LIN {X 0,Y 282.516,Z 595.13,A -85,B 0,C 180,E1 -17100,E2 -17100} C_VEL
LIN {X 0,Y 282.582,Z 591.794,A -85,B 0,C 180,E1 -17102.851,E2 -17102.851} C_VEL
LIN {X 0,Y 282.699,Z 588.163,A -85,B 0,C 180,E1 -17104.992,E2 -17104.992} C_VEL
LIN {X 0,Y 282.973,Z 582.873,A -85,B 0,C 180,E1 -17107.372,E2 -17107.372} C_VEL
LIN {X 0,Y 283.496,Z 576.551,A -85,B 0,C 180,E1 -17109.633,E2 -17109.633} C_VEL
LIN {X 0,Y 284.235,Z 569.125,A -85,B 0,C 180,E1 -17111.771,E2 -17111.771} C_VEL
LIN {X 0,Y 285.228,Z 560.039,A -85,B 0,C 180,E1 -17113.901,E2 -17113.901} C_VEL
LIN {X 0,Y 286.392,Z 549.973,A -85,B 0,C 180,E1 -17115.843,E2 -17115.843} C_VEL
LIN {X 0,Y 287.513,Z 540.083,A -85,B 0,C 180,E1 -17117.419,E2 -17117.419} C_VEL
LIN {X 0,Y 289.014,Z 526.644,A -85,B 0,C 180,E1 -17119.165,E2 -17119.165} C_VEL
LIN {X 0,Y 289.369,Z 520.172,A -85,B 0,C 180,E1 -17119.878,E2 -17119.878} C_VEL
LIN {X 0,Y 287.114,Z 506.341,A -85,B 0,C 180,E1 -17121.272,E2 -17121.272} C_VEL
LIN {X 0,Y 284.752,Z 492.339,A -85,B 0,C 180,E1 -17122.392,E2 -17122.392} C_VEL
LIN {X 0,Y 283.421,Z 484.414,A -85,B 0,C 180,E1 -17122.941,E2 -17122.941} C_VEL
LIN {X 0,Y 283.819,Z 479.195,A -85,B 0,C 180,E1 -17126.942,E2 -17126.942} C_VEL
LIN {X 0,Y 284.155,Z 475.25,A -85,B 0,C 180,E1 -17130.04,E2 -17130.04} C_VEL
LIN {X 0,Y 284.561,Z 470.604,A -85,B 0,C 180,E1 -17133.759,E2 -17133.759} C_VEL
LIN {X 0,Y 284.674,Z 467.49,A -85,B 0,C 180,E1 -17136.336,E2 -17136.336} C_VEL
LIN {X 0,Y 284.462,Z 463.675,A -85,B 0,C 180,E1 -17139.623,E2 -17139.623} C_VEL
LIN {X 0,Y 284.349,Z 463.813,A -85,B 0,C 180,E1 -17141.152,E2 -17141.152} C_VEL
LIN {X 0,Y 285.36,Z 468.719,A -85,B 0,C 180,E1 -17144.418,E2 -17144.418} C_VEL
LIN {X 0,Y 286.241,Z 473.395,A -85,B 0,C 180,E1 -17147.441,E2 -17147.441} C_VEL
LIN {X 0,Y 286.899,Z 478.224,A -85,B 0,C 180,E1 -17150.437,E2 -17150.437} C_VEL
LIN {X 0,Y 286.537,Z 484.384,A -85,B 0,C 180,E1 -17153.937,E2 -17153.937} C_VEL
LIN {X 0,Y 285.97,Z 492.07,A -85,B 0,C 180,E1 -17158.103,E2 -17158.103} C_VEL
LIN {X 0,Y 285.889,Z 493.182,A -85,B 0,C 180,E1 -17158.662,E2 -17158.662} C_VEL
LIN {X 0,Y 290.88,Z 508.242,A -85,B 0,C 180,E1 -17159.827,E2 -17159.827} C_VEL
LIN {X 0,Y 294.37,Z 521.693,A -85,B 0,C 180,E1 -17161.017,E2 -17161.017} C_VEL
LIN {X 0,Y 296.863,Z 535.081,A -85,B 0,C 180,E1 -17162.363,E2 -17162.363} C_VEL
LIN {X 0,Y 297.951,Z 545.247,A -85,B 0,C 180,E1 -17163.511,E2 -17163.511} C_VEL
LIN {X 0,Y 296.029,Z 557.79,A -85,B 0,C 180,E1 -17164.888,E2 -17164.888} C_VEL
LIN {X 0,Y 293.603,Z 570.03,A -85,B 0,C 180,E1 -17166.548,E2 -17166.548} C_VEL
LIN {X 0,Y 291.679,Z 579.114,A -85,B 0,C 180,E1 -17168.068,E2 -17168.068} C_VEL
LIN {X 0,Y 289.463,Z 589.297,A -85,B 0,C 180,E1 -17170.127,E2 -17170.127} C_VEL
LIN {X 0,Y 287.506,Z 597.701,A -85,B 0,C 180,E1 -17172.207,E2 -17172.207} C_VEL
LIN {X 0,Y 285.969,Z 605.714,A -85,B 0,C 180,E1 -17174.679,E2 -17174.679} C_VEL
LIN {X 0,Y 284.396,Z 612.165,A -85,B 0,C 180,E1 -17177.148,E2 -17177.148} C_VEL
LIN {X 0,Y 283.335,Z 617.873,A -85,B 0,C 180,E1 -17179.999,E2 -17179.999} C_VEL
LIN {X 0,Y 282.7,Z 622.021,A -85,B 0,C 180,E1 -17182.858,E2 -17182.858} C_VEL
LIN {X 0,Y 282.371,Z 624.74,A -85,B 0,C 180,E1 -17185.716,E2 -17185.716} C_VEL
LIN {X 0,Y 282.307,Z 626.104,A -85,B 0,C 180,E1 -17188.572,E2 -17188.572} C_VEL
LIN {X 0,Y 282.307,Z 626.137,A -85,B 0,C 180,E1 -17191.425,E2 -17191.425} C_VEL
LIN {X 0,Y 282.369,Z 624.833,A -85,B 0,C 180,E1 -17194.28,E2 -17194.28} C_VEL
LIN {X 0,Y 282.697,Z 622.169,A -85,B 0,C 180,E1 -17197.139,E2 -17197.139} C_VEL
LIN {X 0,Y 283.317,Z 618.072,A -85,B 0,C 180,E1 -17199.998,E2 -17199.998} C_VEL
LIN {X 0,Y 284.328,Z 612.422,A -85,B 0,C 180,E1 -17202.852,E2 -17202.852} C_VEL
LIN {X 0,Y 285.9,Z 606.036,A -85,B 0,C 180,E1 -17205.321,E2 -17205.321} C_VEL
LIN {X 0,Y 287.441,Z 598.344,A -85,B 0,C 180,E1 -17207.72,E2 -17207.72} C_VEL
LIN {X 0,Y 289.392,Z 589.781,A -85,B 0,C 180,E1 -17209.875,E2 -17209.875} C_VEL
LIN {X 0,Y 291.625,Z 579.728,A -85,B 0,C 180,E1 -17211.932,E2 -17211.932} C_VEL
LIN {X 0,Y 293.983,Z 568.473,A -85,B 0,C 180,E1 -17213.79,E2 -17213.79} C_VEL
LIN {X 0,Y 296.157,Z 557.289,A -85,B 0,C 180,E1 -17215.285,E2 -17215.285} C_VEL
LIN {X 0,Y 298.037,Z 545.082,A -85,B 0,C 180,E1 -17216.616,E2 -17216.616} C_VEL
LIN {X 0,Y 296.515,Z 532.609,A -85,B 0,C 180,E1 -17218.007,E2 -17218.007} C_VEL
LIN {X 0,Y 293.649,Z 518.477,A -85,B 0,C 180,E1 -17219.397,E2 -17219.397} C_VEL
LIN {X 0,Y 290.039,Z 505.316,A -85,B 0,C 180,E1 -17220.528,E2 -17220.528} C_VEL
LIN {X 0,Y 285.892,Z 493.075,A -85,B 0,C 180,E1 -17221.49,E2 -17221.49} C_VEL
LIN {X 0,Y 286.527,Z 484.62,A -85,B 0,C 180,E1 -17226.061,E2 -17226.061} C_VEL
LIN {X 0,Y 286.962,Z 478.474,A -85,B 0,C 180,E1 -17229.548,E2 -17229.548} C_VEL
LIN {X 0,Y 286.339,Z 473.573,A -85,B 0,C 180,E1 -17232.58,E2 -17232.58} C_VEL
LIN {X 0,Y 285.25,Z 467.689,A -85,B 0,C 180,E1 -17236.38,E2 -17236.38} C_VEL
LIN {X 0,Y 284.343,Z 463.696,A -85,B 0,C 180,E1 -17239.081,E2 -17239.081} C_VEL
LIN {X 0,Y 284.347,Z 463.691,A -85,B 0,C 180,E1 -17243.616,E2 -17243.616} C_VEL
LIN {X 0,Y 284.301,Z 463.7,A -85,B 0,C 180,E1 -17247.188,E2 -17247.188} C_VEL
LIN {X 0,Y 284.354,Z 463.689,A -85,B 0,C 180,E1 -17250.375,E2 -17250.375} C_VEL
LIN {X 0,Y 284.371,Z 463.676,A -85,B 0,C 180,E1 -17253.586,E2 -17253.586} C_VEL
LIN {X 0,Y 284.366,Z 463.681,A -85,B 0,C 180,E1 -17256.707,E2 -17256.707} C_VEL
LIN {X 0,Y 284.421,Z 463.678,A -85,B 0,C 180,E1 -17259.873,E2 -17259.873} C_VEL
LIN {X 0,Y 284.482,Z 463.671,A -85,B 0,C 180,E1 -17264.458,E2 -17264.458} C_VEL
LIN {X 0,Y 284.48,Z 463.669,A -85,B 0,C 180,E1 -17268.601,E2 -17268.601} C_VEL
LIN {X 0,Y 284.647,Z 463.647,A -85,B 0,C 180,E1 -17271.547,E2 -17271.547} C_VEL
LIN {X 0,Y 283.962,Z 463.739,A -85,B 0,C 180,E1 -17272.726,E2 -17272.726} C_VEL
LIN {X 0,Y 281.114,Z 464.091,A -85,B 0,C 180,E1 -17274.649,E2 -17274.649} C_VEL
LIN {X 0,Y 278.747,Z 464.389,A -85,B 0,C 180,E1 -17276.21,E2 -17276.21} C_VEL
LIN {X 0,Y 277.785,Z 464.506,A -85,B 0,C 180,E1 -17277.419,E2 -17277.419} C_VEL
LIN {X 0,Y 277.735,Z 464.509,A -85,B 0,C 180,E1 -17277.828,E2 -17277.828} C_VEL
LIN {X 0,Y 277.884,Z 464.496,A -85,B 0,C 180,E1 -17280,E2 -17280} C_VEL
LIN {X 0,Y 277.69,Z 464.494,A -85,B 0,C 180,E1 -17282.901,E2 -17282.901} C_VEL
LIN {X 0,Y 277.643,Z 464.526,A -85,B 0,C 180,E1 -17287.271,E2 -17287.271} C_VEL
LIN {X 0,Y 277.497,Z 464.516,A -85,B 0,C 180,E1 -17290.212,E2 -17290.212} C_VEL
LIN {X 0,Y 277.425,Z 464.553,A -85,B 0,C 180,E1 -17294.675,E2 -17294.675} C_VEL
LIN {X 0,Y 277.334,Z 464.554,A -85,B 0,C 180,E1 -17299.234,E2 -17299.234} C_VEL
LIN {X 0,Y 277.31,Z 464.567,A -85,B 0,C 180,E1 -17304.171,E2 -17304.171} C_VEL
LIN {X 0,Y 277.316,Z 464.565,A -85,B 0,C 180,E1 -17307.506,E2 -17307.506} C_VEL
LIN {X 0,Y 277.263,Z 464.572,A -85,B 0,C 180,E1 -17310.482,E2 -17310.482} C_VEL
LIN {X 0,Y 277.246,Z 464.573,A -85,B 0,C 180,E1 -17313.896,E2 -17313.896} C_VEL
LIN {X 0,Y 277.283,Z 464.572,A -85,B 0,C 180,E1 -17317.467,E2 -17317.467} C_VEL
LIN {X 0,Y 277.257,Z 464.571,A -85,B 0,C 180,E1 -17321.228,E2 -17321.228} C_VEL
LIN {X 0,Y 277.308,Z 464.597,A -85,B 0,C 180,E1 -17323.679,E2 -17323.679} C_VEL
LIN {X 0,Y 278.483,Z 471.133,A -85,B 0,C 180,E1 -17328.07,E2 -17328.07} C_VEL
LIN {X 0,Y 279.695,Z 477.445,A -85,B 0,C 180,E1 -17332.088,E2 -17332.088} C_VEL
LIN {X 0,Y 280.717,Z 483.391,A -85,B 0,C 180,E1 -17335.709,E2 -17335.709} C_VEL
LIN {X 0,Y 280.667,Z 484.37,A -85,B 0,C 180,E1 -17336.18,E2 -17336.18} C_VEL
LIN {X 0,Y 280.949,Z 492.018,A -85,B 0,C 180,E1 -17338.069,E2 -17338.069} C_VEL
LIN {X 0,Y 285.484,Z 507.635,A -85,B 0,C 180,E1 -17339.137,E2 -17339.137} C_VEL
LIN {X 0,Y 288.26,Z 521.704,A -85,B 0,C 180,E1 -17340.206,E2 -17340.206} C_VEL
LIN {X 0,Y 290.029,Z 534.468,A -85,B 0,C 180,E1 -17341.351,E2 -17341.351} C_VEL
LIN {X 0,Y 291.046,Z 547.26,A -85,B 0,C 180,E1 -17342.693,E2 -17342.693} C_VEL
LIN {X 0,Y 290.475,Z 552.892,A -85,B 0,C 180,E1 -17343.276,E2 -17343.276} C_VEL
LIN {X 0,Y 288.548,Z 564.116,A -85,B 0,C 180,E1 -17344.577,E2 -17344.577} C_VEL
LIN {X 0,Y 286.145,Z 576.029,A -85,B 0,C 180,E1 -17346.287,E2 -17346.287} C_VEL
LIN {X 0,Y 283.762,Z 586.747,A -85,B 0,C 180,E1 -17348.193,E2 -17348.193} C_VEL
LIN {X 0,Y 281.559,Z 596.39,A -85,B 0,C 180,E1 -17350.31,E2 -17350.31} C_VEL
LIN {X 0,Y 279.68,Z 604.372,A -85,B 0,C 180,E1 -17352.452,E2 -17352.452} C_VEL
LIN {X 0,Y 278.313,Z 611.004,A -85,B 0,C 180,E1 -17354.626,E2 -17354.626} C_VEL
LIN {X 0,Y 277.137,Z 616.5,A -85,B 0,C 180,E1 -17356.809,E2 -17356.809} C_VEL
LIN {X 0,Y 276.088,Z 622.251,A -85,B 0,C 180,E1 -17359.738,E2 -17359.738} C_VEL
LIN {X 0,Y 275.484,Z 626.427,A -85,B 0,C 180,E1 -17362.673,E2 -17362.673} C_VEL
LIN {X 0,Y 275.242,Z 629.15,A -85,B 0,C 180,E1 -17365.609,E2 -17365.609} C_VEL
LIN {X 0,Y 275.26,Z 630.498,A -85,B 0,C 180,E1 -17368.539,E2 -17368.539} C_VEL
LIN {X 0,Y 275.262,Z 630.49,A -85,B 0,C 180,E1 -17371.465,E2 -17371.465} C_VEL
LIN {X 0,Y 275.245,Z 629.125,A -85,B 0,C 180,E1 -17374.395,E2 -17374.395} C_VEL
LIN {X 0,Y 275.487,Z 626.388,A -85,B 0,C 180,E1 -17377.33,E2 -17377.33} C_VEL
LIN {X 0,Y 276.087,Z 622.203,A -85,B 0,C 180,E1 -17380.266,E2 -17380.266} C_VEL
LIN {X 0,Y 277.129,Z 616.438,A -85,B 0,C 180,E1 -17383.195,E2 -17383.195} C_VEL
LIN {X 0,Y 278.358,Z 611.305,A -85,B 0,C 180,E1 -17385.375,E2 -17385.375} C_VEL
LIN {X 0,Y 280.569,Z 605.09,A -85,B 0,C 180,E1 -17388.249,E2 -17388.249} C_VEL
LIN {X 0,Y 283.729,Z 597.292,A -85,B 0,C 180,E1 -17391.051,E2 -17391.051} C_VEL
LIN {X 0,Y 287.043,Z 589.043,A -85,B 0,C 180,E1 -17393.447,E2 -17393.447} C_VEL
LIN {X 0,Y 291.101,Z 579.224,A -85,B 0,C 180,E1 -17395.76,E2 -17395.76} C_VEL
LIN {X 0,Y 295.088,Z 569.27,A -85,B 0,C 180,E1 -17397.675,E2 -17397.675} C_VEL
LIN {X 0,Y 299.923,Z 556.493,A -85,B 0,C 180,E1 -17399.672,E2 -17399.672} C_VEL
LIN {X 0,Y 300.93,Z 552.397,A -85,B 0,C 180,E1 -17400.335,E2 -17400.335} C_VEL
LIN {X 0,Y 301.69,Z 544.958,A -85,B 0,C 180,E1 -17401.704,E2 -17401.704} C_VEL
LIN {X 0,Y 301.702,Z 535.626,A -85,B 0,C 180,E1 -17403.603,E2 -17403.603} C_VEL
LIN {X 0,Y 300.973,Z 526.547,A -85,B 0,C 180,E1 -17405.718,E2 -17405.718} C_VEL
LIN {X 0,Y 299.975,Z 521.596,A -85,B 0,C 180,E1 -17407.196,E2 -17407.196} C_VEL
LIN {X 0,Y 298.426,Z 517.301,A -85,B 0,C 180,E1 -17408.999,E2 -17408.999} C_VEL
LIN {X 0,Y 296.626,Z 512.895,A -85,B 0,C 180,E1 -17411.562,E2 -17411.562} C_VEL
LIN {X 0,Y 295.198,Z 510.586,A -85,B 0,C 180,E1 -17414.42,E2 -17414.42} C_VEL
LIN {X 0,Y 294.84,Z 509.961,A -85,B 0,C 180,E1 -17416.27,E2 -17416.27} C_VEL
LIN {X 0,Y 294.99,Z 509.937,A -85,B 0,C 180,E1 -17418.157,E2 -17418.157} C_VEL
LIN {X 0,Y 295.651,Z 510.537,A -85,B 0,C 180,E1 -17420.072,E2 -17420.072} C_VEL
LIN {X 0,Y 296.715,Z 513.686,A -85,B 0,C 180,E1 -17422.672,E2 -17422.672} C_VEL
LIN {X 0,Y 297.338,Z 515.534,A -85,B 0,C 180,E1 -17423.778,E2 -17423.778} C_VEL
LIN {X 0,Y 298.913,Z 521.216,A -85,B 0,C 180,E1 -17426.347,E2 -17426.347} C_VEL
LIN {X 0,Y 300.321,Z 527.635,A -85,B 0,C 180,E1 -17428.584,E2 -17428.584} C_VEL
LIN {X 0,Y 301.365,Z 535.546,A -85,B 0,C 180,E1 -17430.874,E2 -17430.874} C_VEL
LIN {X 0,Y 301.588,Z 542.791,A -85,B 0,C 180,E1 -17432.712,E2 -17432.712} C_VEL
LIN {X 0,Y 301.478,Z 544.356,A -85,B 0,C 180,E1 -17433.076,E2 -17433.076} C_VEL
LIN {X 0,Y 297.491,Z 554.629,A -85,B 0,C 180,E1 -17434.834,E2 -17434.834} C_VEL
LIN {X 0,Y 293.555,Z 563.94,A -85,B 0,C 180,E1 -17436.732,E2 -17436.732} C_VEL
LIN {X 0,Y 289.465,Z 572.864,A -85,B 0,C 180,E1 -17439.015,E2 -17439.015} C_VEL
LIN {X 0,Y 286.819,Z 578.347,A -85,B 0,C 180,E1 -17440.683,E2 -17440.683} C_VEL
LIN {X 0,Y 283.411,Z 585.379,A -85,B 0,C 180,E1 -17443.431,E2 -17443.431} C_VEL
LIN {X 0,Y 281.353,Z 589.557,A -85,B 0,C 180,E1 -17445.535,E2 -17445.535} C_VEL
LIN {X 0,Y 279.983,Z 591.874,A -85,B 0,C 180,E1 -17446.943,E2 -17446.943} C_VEL
LIN {X 0,Y 278.229,Z 595.227,A -85,B 0,C 180,E1 -17449.816,E2 -17449.816} C_VEL
LIN {X 0,Y 276.731,Z 597.123,A -85,B 0,C 180,E1 -17452.705,E2 -17452.705} C_VEL
LIN {X 0,Y 275.956,Z 597.527,A -85,B 0,C 180,E1 -17455.618,E2 -17455.618} C_VEL
LIN {X 0,Y 275.72,Z 597.15,A -85,B 0,C 180,E1 -17457.078,E2 -17457.078} C_VEL
LIN {X 0,Y 275.432,Z 595.211,A -85,B 0,C 180,E1 -17460,E2 -17460} C_VEL
LIN {X 0,Y 275.512,Z 591.717,A -85,B 0,C 180,E1 -17462.924,E2 -17462.924} C_VEL
LIN {X 0,Y 275.604,Z 587.935,A -85,B 0,C 180,E1 -17465.121,E2 -17465.121} C_VEL
LIN {X 0,Y 275.877,Z 582.801,A -85,B 0,C 180,E1 -17467.422,E2 -17467.422} C_VEL
LIN {X 0,Y 276.484,Z 575.876,A -85,B 0,C 180,E1 -17469.88,E2 -17469.88} C_VEL
LIN {X 0,Y 277.254,Z 568.235,A -85,B 0,C 180,E1 -17472.071,E2 -17472.071} C_VEL
LIN {X 0,Y 278.303,Z 558.977,A -85,B 0,C 180,E1 -17474.254,E2 -17474.254} C_VEL
LIN {X 0,Y 279.694,Z 547.592,A -85,B 0,C 180,E1 -17476.421,E2 -17476.421} C_VEL
LIN {X 0,Y 280.994,Z 535.882,A -85,B 0,C 180,E1 -17478.231,E2 -17478.231} C_VEL
LIN {X 0,Y 282.357,Z 522.98,A -85,B 0,C 180,E1 -17479.824,E2 -17479.824} C_VEL
LIN {X 0,Y 282.066,Z 519.454,A -85,B 0,C 180,E1 -17480.225,E2 -17480.225} C_VEL
LIN {X 0,Y 279.821,Z 505.317,A -85,B 0,C 180,E1 -17481.671,E2 -17481.671} C_VEL
LIN {X 0,Y 277.293,Z 490.17,A -85,B 0,C 180,E1 -17482.879,E2 -17482.879} C_VEL
LIN {X 0,Y 276.342,Z 484.556,A -85,B 0,C 180,E1 -17483.27,E2 -17483.27} C_VEL
LIN {X 0,Y 276.777,Z 479.447,A -85,B 0,C 180,E1 -17487.283,E2 -17487.283} C_VEL
LIN {X 0,Y 277.249,Z 474.438,A -85,B 0,C 180,E1 -17491.309,E2 -17491.309} C_VEL
LIN {X 0,Y 277.508,Z 471.327,A -85,B 0,C 180,E1 -17493.86,E2 -17493.86} C_VEL
LIN {X 0,Y 277.617,Z 467.126,A -85,B 0,C 180,E1 -17497.414,E2 -17497.414} C_VEL
LIN {X 0,Y 277.417,Z 464.552,A -85,B 0,C 180,E1 -17499.745,E2 -17499.745} C_VEL
LIN {X 0,Y 277.387,Z 464.764,A -85,B 0,C 180,E1 -17500.386,E2 -17500.386} C_VEL
LIN {X 0,Y 278.403,Z 469.972,A -85,B 0,C 180,E1 -17503.965,E2 -17503.965} C_VEL
LIN {X 0,Y 279.571,Z 476.393,A -85,B 0,C 180,E1 -17508.169,E2 -17508.169} C_VEL
LIN {X 0,Y 280.004,Z 481.093,A -85,B 0,C 180,E1 -17511.086,E2 -17511.086} C_VEL
LIN {X 0,Y 279.492,Z 487.386,A -85,B 0,C 180,E1 -17514.664,E2 -17514.664} C_VEL
LIN {X 0,Y 279.058,Z 493.172,A -85,B 0,C 180,E1 -17517.806,E2 -17517.806} C_VEL
LIN {X 0,Y 284.232,Z 508.512,A -85,B 0,C 180,E1 -17519.058,E2 -17519.058} C_VEL
LIN {X 0,Y 287.63,Z 521.539,A -85,B 0,C 180,E1 -17520.258,E2 -17520.258} C_VEL
LIN {X 0,Y 289.979,Z 533.81,A -85,B 0,C 180,E1 -17521.53,E2 -17521.53} C_VEL
LIN {X 0,Y 291.387,Z 545.201,A -85,B 0,C 180,E1 -17522.856,E2 -17522.856} C_VEL
LIN {X 0,Y 290.471,Z 552.809,A -85,B 0,C 180,E1 -17523.688,E2 -17523.688} C_VEL
LIN {X 0,Y 288.35,Z 564.29,A -85,B 0,C 180,E1 -17525.136,E2 -17525.136} C_VEL
LIN {X 0,Y 285.884,Z 575.326,A -85,B 0,C 180,E1 -17526.836,E2 -17526.836} C_VEL
LIN {X 0,Y 283.557,Z 586.15,A -85,B 0,C 180,E1 -17528.936,E2 -17528.936} C_VEL
LIN {X 0,Y 281.379,Z 595.089,A -85,B 0,C 180,E1 -17531.051,E2 -17531.051} C_VEL
LIN {X 0,Y 279.653,Z 602.529,A -85,B 0,C 180,E1 -17533.2,E2 -17533.2} C_VEL
LIN {X 0,Y 278.33,Z 608.729,A -85,B 0,C 180,E1 -17535.372,E2 -17535.372} C_VEL
LIN {X 0,Y 277.134,Z 613.813,A -85,B 0,C 180,E1 -17537.55,E2 -17537.55} C_VEL
LIN {X 0,Y 276.116,Z 619.138,A -85,B 0,C 180,E1 -17540.475,E2 -17540.475} C_VEL
LIN {X 0,Y 275.631,Z 622.077,A -85,B 0,C 180,E1 -17542.674,E2 -17542.674} C_VEL
LIN {X 0,Y 275.285,Z 624.796,A -85,B 0,C 180,E1 -17545.606,E2 -17545.606} C_VEL
LIN {X 0,Y 275.234,Z 626.159,A -85,B 0,C 180,E1 -17548.535,E2 -17548.535} C_VEL
LIN {X 0,Y 275.234,Z 626.192,A -85,B 0,C 180,E1 -17551.461,E2 -17551.461} C_VEL
LIN {X 0,Y 275.282,Z 624.888,A -85,B 0,C 180,E1 -17554.391,E2 -17554.391} C_VEL
LIN {X 0,Y 275.628,Z 622.223,A -85,B 0,C 180,E1 -17557.323,E2 -17557.323} C_VEL
LIN {X 0,Y 276.285,Z 618.126,A -85,B 0,C 180,E1 -17560.255,E2 -17560.255} C_VEL
LIN {X 0,Y 277.378,Z 612.475,A -85,B 0,C 180,E1 -17563.179,E2 -17563.179} C_VEL
LIN {X 0,Y 279.026,Z 606.088,A -85,B 0,C 180,E1 -17565.708,E2 -17565.708} C_VEL
LIN {X 0,Y 280.639,Z 598.394,A -85,B 0,C 180,E1 -17568.165,E2 -17568.165} C_VEL
LIN {X 0,Y 282.719,Z 589.829,A -85,B 0,C 180,E1 -17570.364,E2 -17570.364} C_VEL
LIN {X 0,Y 285.028,Z 579.773,A -85,B 0,C 180,E1 -17572.467,E2 -17572.467} C_VEL
LIN {X 0,Y 287.496,Z 568.514,A -85,B 0,C 180,E1 -17574.361,E2 -17574.361} C_VEL
LIN {X 0,Y 289.949,Z 556.086,A -85,B 0,C 180,E1 -17576.037,E2 -17576.037} C_VEL
LIN {X 0,Y 291.501,Z 546.583,A -85,B 0,C 180,E1 -17577.095,E2 -17577.095} C_VEL
LIN {X 0,Y 290.271,Z 535.149,A -85,B 0,C 180,E1 -17578.436,E2 -17578.436} C_VEL
LIN {X 0,Y 287.743,Z 521.887,A -85,B 0,C 180,E1 -17579.825,E2 -17579.825} C_VEL
LIN {X 0,Y 284.306,Z 508.566,A -85,B 0,C 180,E1 -17581.053,E2 -17581.053} C_VEL
LIN {X 0,Y 279.722,Z 495.37,A -85,B 0,C 180,E1 -17582.167,E2 -17582.167} C_VEL
LIN {X 0,Y 279.056,Z 493.021,A -85,B 0,C 180,E1 -17582.385,E2 -17582.385} C_VEL
LIN {X 0,Y 279.641,Z 485.63,A -85,B 0,C 180,E1 -17586.464,E2 -17586.464} C_VEL
LIN {X 0,Y 280.06,Z 479.893,A -85,B 0,C 180,E1 -17589.782,E2 -17589.782} C_VEL
LIN {X 0,Y 279.425,Z 475.143,A -85,B 0,C 180,E1 -17592.77,E2 -17592.77} C_VEL
LIN {X 0,Y 278.513,Z 470.142,A -85,B 0,C 180,E1 -17596.057,E2 -17596.057} C_VEL
LIN {X 0,Y 277.298,Z 464.567,A -85,B 0,C 180,E1 -17599.955,E2 -17599.955} C_VEL
LIN {X 0,Y 277.298,Z 464.569,A -85,B 0,C 180,E1 -17604.343,E2 -17604.343} C_VEL
LIN {X 0,Y 277.238,Z 464.575,A -85,B 0,C 180,E1 -17607.835,E2 -17607.835} C_VEL
LIN {X 0,Y 277.297,Z 464.572,A -85,B 0,C 180,E1 -17611.213,E2 -17611.213} C_VEL
LIN {X 0,Y 277.311,Z 464.562,A -85,B 0,C 180,E1 -17614.479,E2 -17614.479} C_VEL
LIN {X 0,Y 277.284,Z 464.554,A -85,B 0,C 180,E1 -17617.655,E2 -17617.655} C_VEL
LIN {X 0,Y 277.364,Z 464.561,A -85,B 0,C 180,E1 -17620.767,E2 -17620.767} C_VEL
LIN {X 0,Y 277.425,Z 464.549,A -85,B 0,C 180,E1 -17625.325,E2 -17625.325} C_VEL
LIN {X 0,Y 277.497,Z 464.544,A -85,B 0,C 180,E1 -17629.788,E2 -17629.788} C_VEL
LIN {X 0,Y 277.644,Z 464.526,A -85,B 0,C 180,E1 -17632.729,E2 -17632.729} C_VEL
LIN {X 0,Y 277.735,Z 464.509,A -85,B 0,C 180,E1 -17637.828,E2 -17637.828} C_VEL
LIN {X 0,Y 277.13,Z 464.586,A -85,B 0,C 180,E1 -17639.04,E2 -17639.04} C_VEL
LIN {X 0,Y 274.239,Z 464.947,A -85,B 0,C 180,E1 -17641.01,E2 -17641.01} C_VEL
LIN {X 0,Y 271.699,Z 465.246,A -85,B 0,C 180,E1 -17642.611,E2 -17642.611} C_VEL
LIN {X 0,Y 270.551,Z 465.38,A -85,B 0,C 180,E1 -17643.854,E2 -17643.854} C_VEL
LIN {X 0,Y 270.43,Z 465.396,A -85,B 0,C 180,E1 -17644.277,E2 -17644.277} C_VEL
LIN {X 0,Y 270.601,Z 465.403,A -85,B 0,C 180,E1 -17647.461,E2 -17647.461} C_VEL
LIN {X 0,Y 270.432,Z 465.395,A -85,B 0,C 180,E1 -17650.481,E2 -17650.481} C_VEL
LIN {X 0,Y 270.393,Z 465.425,A -85,B 0,C 180,E1 -17655.065,E2 -17655.065} C_VEL
LIN {X 0,Y 270.291,Z 465.438,A -85,B 0,C 180,E1 -17659.756,E2 -17659.756} C_VEL
LIN {X 0,Y 270.265,Z 465.444,A -85,B 0,C 180,E1 -17664.586,E2 -17664.586} C_VEL
LIN {X 0,Y 270.263,Z 465.442,A -85,B 0,C 180,E1 -17667.91,E2 -17667.91} C_VEL
LIN {X 0,Y 270.176,Z 465.453,A -85,B 0,C 180,E1 -17671.349,E2 -17671.349} C_VEL
LIN {X 0,Y 270.208,Z 465.454,A -85,B 0,C 180,E1 -17674.905,E2 -17674.905} C_VEL
LIN {X 0,Y 270.214,Z 465.449,A -85,B 0,C 180,E1 -17678.718,E2 -17678.718} C_VEL
LIN {X 0,Y 270.223,Z 465.452,A -85,B 0,C 180,E1 -17682.548,E2 -17682.548} C_VEL
LIN {X 0,Y 270.282,Z 465.661,A -85,B 0,C 180,E1 -17683.498,E2 -17683.498} C_VEL
LIN {X 0,Y 271.374,Z 471.715,A -85,B 0,C 180,E1 -17687.677,E2 -17687.677} C_VEL
LIN {X 0,Y 272.597,Z 477.954,A -85,B 0,C 180,E1 -17691.777,E2 -17691.777} C_VEL
LIN {X 0,Y 273.419,Z 482.413,A -85,B 0,C 180,E1 -17694.579,E2 -17694.579} C_VEL
LIN {X 0,Y 274.17,Z 486.192,A -85,B 0,C 180,E1 -17695.674,E2 -17695.674} C_VEL
LIN {X 0,Y 274.3,Z 491.913,A -85,B 0,C 180,E1 -17697.179,E2 -17697.179} C_VEL
LIN {X 0,Y 279.021,Z 507.885,A -85,B 0,C 180,E1 -17698.35,E2 -17698.35} C_VEL
LIN {X 0,Y 281.839,Z 521.875,A -85,B 0,C 180,E1 -17699.467,E2 -17699.467} C_VEL
LIN {X 0,Y 283.653,Z 535.636,A -85,B 0,C 180,E1 -17700.753,E2 -17700.753} C_VEL
LIN {X 0,Y 284.597,Z 548.982,A -85,B 0,C 180,E1 -17702.22,E2 -17702.22} C_VEL
LIN {X 0,Y 283.137,Z 558.542,A -85,B 0,C 180,E1 -17703.265,E2 -17703.265} C_VEL
LIN {X 0,Y 280.879,Z 570.345,A -85,B 0,C 180,E1 -17704.829,E2 -17704.829} C_VEL
LIN {X 0,Y 278.458,Z 581.117,A -85,B 0,C 180,E1 -17706.579,E2 -17706.579} C_VEL
LIN {X 0,Y 275.963,Z 591.753,A -85,B 0,C 180,E1 -17708.723,E2 -17708.723} C_VEL
LIN {X 0,Y 273.812,Z 600.516,A -85,B 0,C 180,E1 -17710.9,E2 -17710.9} C_VEL
LIN {X 0,Y 271.867,Z 608.903,A -85,B 0,C 180,E1 -17713.482,E2 -17713.482} C_VEL
LIN {X 0,Y 270.611,Z 614.733,A -85,B 0,C 180,E1 -17715.718,E2 -17715.718} C_VEL
LIN {X 0,Y 269.271,Z 620.946,A -85,B 0,C 180,E1 -17718.713,E2 -17718.713} C_VEL
LIN {X 0,Y 268.681,Z 624.473,A -85,B 0,C 180,E1 -17720.972,E2 -17720.972} C_VEL
LIN {X 0,Y 268.253,Z 627.909,A -85,B 0,C 180,E1 -17723.987,E2 -17723.987} C_VEL
LIN {X 0,Y 268.165,Z 629.938,A -85,B 0,C 180,E1 -17726.997,E2 -17726.997} C_VEL
LIN {X 0,Y 268.186,Z 630.442,A -85,B 0,C 180,E1 -17728.5,E2 -17728.5} C_VEL
LIN {X 0,Y 268.188,Z 630.434,A -85,B 0,C 180,E1 -17731.504,E2 -17731.504} C_VEL
LIN {X 0,Y 268.165,Z 629.069,A -85,B 0,C 180,E1 -17734.511,E2 -17734.511} C_VEL
LIN {X 0,Y 268.408,Z 626.332,A -85,B 0,C 180,E1 -17737.525,E2 -17737.525} C_VEL
LIN {X 0,Y 269.047,Z 622.147,A -85,B 0,C 180,E1 -17740.538,E2 -17740.538} C_VEL
LIN {X 0,Y 270.201,Z 616.383,A -85,B 0,C 180,E1 -17743.54,E2 -17743.54} C_VEL
LIN {X 0,Y 271.046,Z 612.911,A -85,B 0,C 180,E1 -17745.03,E2 -17745.03} C_VEL
LIN {X 0,Y 273.151,Z 607.333,A -85,B 0,C 180,E1 -17747.986,E2 -17747.986} C_VEL
LIN {X 0,Y 276.312,Z 600.265,A -85,B 0,C 180,E1 -17750.862,E2 -17750.862} C_VEL
LIN {X 0,Y 279.547,Z 592.769,A -85,B 0,C 180,E1 -17753.328,E2 -17753.328} C_VEL
LIN {X 0,Y 283.647,Z 583.809,A -85,B 0,C 180,E1 -17755.698,E2 -17755.698} C_VEL
LIN {X 0,Y 288.319,Z 573.166,A -85,B 0,C 180,E1 -17757.986,E2 -17757.986} C_VEL
LIN {X 0,Y 293.281,Z 561.401,A -85,B 0,C 180,E1 -17760.013,E2 -17760.013} C_VEL
LIN {X 0,Y 294.87,Z 557.373,A -85,B 0,C 180,E1 -17760.629,E2 -17760.629} C_VEL
LIN {X 0,Y 296.134,Z 551.129,A -85,B 0,C 180,E1 -17761.785,E2 -17761.785} C_VEL
LIN {X 0,Y 296.765,Z 542.324,A -85,B 0,C 180,E1 -17763.645,E2 -17763.645} C_VEL
LIN {X 0,Y 296.762,Z 533.966,A -85,B 0,C 180,E1 -17765.584,E2 -17765.584} C_VEL
LIN {X 0,Y 296.404,Z 529.254,A -85,B 0,C 180,E1 -17766.879,E2 -17766.879} C_VEL
LIN {X 0,Y 295.533,Z 525.381,A -85,B 0,C 180,E1 -17768.301,E2 -17768.301} C_VEL
LIN {X 0,Y 294.977,Z 523.622,A -85,B 0,C 180,E1 -17769.101,E2 -17769.101} C_VEL
LIN {X 0,Y 293.131,Z 518.714,A -85,B 0,C 180,E1 -17772.171,E2 -17772.171} C_VEL
LIN {X 0,Y 292.262,Z 517.149,A -85,B 0,C 180,E1 -17774.218,E2 -17774.218} C_VEL
LIN {X 0,Y 291.846,Z 516.395,A -85,B 0,C 180,E1 -17776.258,E2 -17776.258} C_VEL
LIN {X 0,Y 291.975,Z 516.365,A -85,B 0,C 180,E1 -17778.263,E2 -17778.263} C_VEL
LIN {X 0,Y 292.348,Z 516.677,A -85,B 0,C 180,E1 -17779.528,E2 -17779.528} C_VEL
LIN {X 0,Y 292.841,Z 518.429,A -85,B 0,C 180,E1 -17781.392,E2 -17781.392} C_VEL
LIN {X 0,Y 293.633,Z 520.968,A -85,B 0,C 180,E1 -17783.247,E2 -17783.247} C_VEL
LIN {X 0,Y 294.693,Z 526.193,A -85,B 0,C 180,E1 -17785.768,E2 -17785.768} C_VEL
LIN {X 0,Y 295.67,Z 532.175,A -85,B 0,C 180,E1 -17788.032,E2 -17788.032} C_VEL
LIN {X 0,Y 296.293,Z 540.408,A -85,B 0,C 180,E1 -17790.566,E2 -17790.566} C_VEL
LIN {X 0,Y 296.112,Z 546.922,A -85,B 0,C 180,E1 -17792.303,E2 -17792.303} C_VEL
LIN {X 0,Y 290.795,Z 559.359,A -85,B 0,C 180,E1 -17794.597,E2 -17794.597} C_VEL
LIN {X 0,Y 286.14,Z 569.117,A -85,B 0,C 180,E1 -17796.86,E2 -17796.86} C_VEL
LIN {X 0,Y 281.972,Z 577.226,A -85,B 0,C 180,E1 -17799.196,E2 -17799.196} C_VEL
LIN {X 0,Y 278.534,Z 583.778,A -85,B 0,C 180,E1 -17801.615,E2 -17801.615} C_VEL
LIN {X 0,Y 276.012,Z 588.318,A -85,B 0,C 180,E1 -17803.735,E2 -17803.735} C_VEL
LIN {X 0,Y 273.175,Z 592.981,A -85,B 0,C 180,E1 -17806.612,E2 -17806.612} C_VEL
LIN {X 0,Y 271.299,Z 596.068,A -85,B 0,C 180,E1 -17809.553,E2 -17809.553} C_VEL
LIN {X 0,Y 269.739,Z 597.742,A -85,B 0,C 180,E1 -17812.515,E2 -17812.515} C_VEL
LIN {X 0,Y 269.222,Z 598.017,A -85,B 0,C 180,E1 -17814.006,E2 -17814.006} C_VEL
LIN {X 0,Y 268.648,Z 597.397,A -85,B 0,C 180,E1 -17817.001,E2 -17817.001} C_VEL
LIN {X 0,Y 268.349,Z 595.282,A -85,B 0,C 180,E1 -17820,E2 -17820} C_VEL
LIN {X 0,Y 268.369,Z 592.624,A -85,B 0,C 180,E1 -17822.251,E2 -17822.251} C_VEL
LIN {X 0,Y 268.48,Z 589.017,A -85,B 0,C 180,E1 -17824.504,E2 -17824.504} C_VEL
LIN {X 0,Y 268.69,Z 584.37,A -85,B 0,C 180,E1 -17826.759,E2 -17826.759} C_VEL
LIN {X 0,Y 269.223,Z 577.507,A -85,B 0,C 180,E1 -17829.39,E2 -17829.39} C_VEL
LIN {X 0,Y 269.966,Z 570.125,A -85,B 0,C 180,E1 -17831.64,E2 -17831.64} C_VEL
LIN {X 0,Y 270.923,Z 561.133,A -85,B 0,C 180,E1 -17833.884,E2 -17833.884} C_VEL
LIN {X 0,Y 272.006,Z 552.182,A -85,B 0,C 180,E1 -17835.742,E2 -17835.742} C_VEL
LIN {X 0,Y 273.205,Z 542.673,A -85,B 0,C 180,E1 -17837.4,E2 -17837.4} C_VEL
LIN {X 0,Y 274.464,Z 531.303,A -85,B 0,C 180,E1 -17839.055,E2 -17839.055} C_VEL
LIN {X 0,Y 275.374,Z 522.267,A -85,B 0,C 180,E1 -17840.154,E2 -17840.154} C_VEL
LIN {X 0,Y 273.28,Z 509.142,A -85,B 0,C 180,E1 -17841.589,E2 -17841.589} C_VEL
LIN {X 0,Y 271.056,Z 495.449,A -85,B 0,C 180,E1 -17842.801,E2 -17842.801} C_VEL
LIN {X 0,Y 269.276,Z 484.781,A -85,B 0,C 180,E1 -17843.565,E2 -17843.565} C_VEL
LIN {X 0,Y 269.776,Z 479.287,A -85,B 0,C 180,E1 -17847.965,E2 -17847.965} C_VEL
LIN {X 0,Y 270.328,Z 474.134,A -85,B 0,C 180,E1 -17852.206,E2 -17852.206} C_VEL
LIN {X 0,Y 270.508,Z 470.993,A -85,B 0,C 180,E1 -17854.86,E2 -17854.86} C_VEL
LIN {X 0,Y 270.514,Z 466.498,A -85,B 0,C 180,E1 -17858.792,E2 -17858.792} C_VEL
LIN {X 0,Y 270.436,Z 465.74,A -85,B 0,C 180,E1 -17859.588,E2 -17859.588} C_VEL
LIN {X 0,Y 271.692,Z 472.458,A -85,B 0,C 180,E1 -17864.301,E2 -17864.301} C_VEL
LIN {X 0,Y 272.755,Z 478.528,A -85,B 0,C 180,E1 -17868.352,E2 -17868.352} C_VEL
LIN {X 0,Y 273.109,Z 482.004,A -85,B 0,C 180,E1 -17870.534,E2 -17870.534} C_VEL
LIN {X 0,Y 272.732,Z 487.314,A -85,B 0,C 180,E1 -17873.65,E2 -17873.65} C_VEL
LIN {X 0,Y 272.224,Z 493.14,A -85,B 0,C 180,E1 -17876.896,E2 -17876.896} C_VEL
LIN {X 0,Y 277.306,Z 507.86,A -85,B 0,C 180,E1 -17878.163,E2 -17878.163} C_VEL
LIN {X 0,Y 280.881,Z 521.038,A -85,B 0,C 180,E1 -17879.431,E2 -17879.431} C_VEL
LIN {X 0,Y 283.395,Z 533.846,A -85,B 0,C 180,E1 -17880.806,E2 -17880.806} C_VEL
LIN {X 0,Y 284.932,Z 546.612,A -85,B 0,C 180,E1 -17882.347,E2 -17882.347} C_VEL
LIN {X 0,Y 283.192,Z 557.882,A -85,B 0,C 180,E1 -17883.664,E2 -17883.664} C_VEL
LIN {X 0,Y 280.63,Z 570.129,A -85,B 0,C 180,E1 -17885.394,E2 -17885.394} C_VEL
LIN {X 0,Y 278.521,Z 579.217,A -85,B 0,C 180,E1 -17886.974,E2 -17886.974} C_VEL
LIN {X 0,Y 276.131,Z 589.403,A -85,B 0,C 180,E1 -17889.124,E2 -17889.124} C_VEL
LIN {X 0,Y 273.975,Z 597.807,A -85,B 0,C 180,E1 -17891.296,E2 -17891.296} C_VEL
LIN {X 0,Y 272.429,Z 604.783,A -85,B 0,C 180,E1 -17893.513,E2 -17893.513} C_VEL
LIN {X 0,Y 270.966,Z 610.57,A -85,B 0,C 180,E1 -17895.734,E2 -17895.734} C_VEL
LIN {X 0,Y 269.567,Z 616.741,A -85,B 0,C 180,E1 -17898.722,E2 -17898.722} C_VEL
LIN {X 0,Y 268.888,Z 620.245,A -85,B 0,C 180,E1 -17900.976,E2 -17900.976} C_VEL
LIN {X 0,Y 268.348,Z 623.666,A -85,B 0,C 180,E1 -17903.985,E2 -17903.985} C_VEL
LIN {X 0,Y 268.174,Z 625.7,A -85,B 0,C 180,E1 -17906.994,E2 -17906.994} C_VEL
LIN {X 0,Y 268.146,Z 626.398,A -85,B 0,C 180,E1 -17909.998,E2 -17909.998} C_VEL
LIN {X 0,Y 268.173,Z 625.764,A -85,B 0,C 180,E1 -17913.003,E2 -17913.003} C_VEL
LIN {X 0,Y 268.347,Z 623.784,A -85,B 0,C 180,E1 -17916.011,E2 -17916.011} C_VEL
LIN {X 0,Y 268.882,Z 620.415,A -85,B 0,C 180,E1 -17919.021,E2 -17919.021} C_VEL
LIN {X 0,Y 269.806,Z 615.557,A -85,B 0,C 180,E1 -17922.026,E2 -17922.026} C_VEL
LIN {X 0,Y 270.918,Z 610.852,A -85,B 0,C 180,E1 -17924.265,E2 -17924.265} C_VEL
LIN {X 0,Y 272.323,Z 605.131,A -85,B 0,C 180,E1 -17926.49,E2 -17926.49} C_VEL
LIN {X 0,Y 274.243,Z 596.898,A -85,B 0,C 180,E1 -17929.069,E2 -17929.069} C_VEL
LIN {X 0,Y 276.462,Z 588.308,A -85,B 0,C 180,E1 -17931.236,E2 -17931.236} C_VEL
LIN {X 0,Y 278.891,Z 577.9,A -85,B 0,C 180,E1 -17933.382,E2 -17933.382} C_VEL
LIN {X 0,Y 281.306,Z 567.404,A -85,B 0,C 180,E1 -17935.131,E2 -17935.131} C_VEL
LIN {X 0,Y 283.654,Z 555.654,A -85,B 0,C 180,E1 -17936.727,E2 -17936.727} C_VEL
LIN {X 0,Y 284.934,Z 548.289,A -85,B 0,C 180,E1 -17937.572,E2 -17937.572} C_VEL
LIN {X 0,Y 283.998,Z 537.611,A -85,B 0,C 180,E1 -17938.874,E2 -17938.874} C_VEL
LIN {X 0,Y 281.602,Z 524.239,A -85,B 0,C 180,E1 -17940.365,E2 -17940.365} C_VEL
LIN {X 0,Y 278.384,Z 511.113,A -85,B 0,C 180,E1 -17941.652,E2 -17941.652} C_VEL
LIN {X 0,Y 273.729,Z 497.31,A -85,B 0,C 180,E1 -17942.894,E2 -17942.894} C_VEL
LIN {X 0,Y 272.234,Z 493.074,A -85,B 0,C 180,E1 -17943.274,E2 -17943.274} C_VEL
LIN {X 0,Y 272.791,Z 486.47,A -85,B 0,C 180,E1 -17946.997,E2 -17946.997} C_VEL
LIN {X 0,Y 273.172,Z 481.309,A -85,B 0,C 180,E1 -17950.027,E2 -17950.027} C_VEL
LIN {X 0,Y 272.569,Z 476.838,A -85,B 0,C 180,E1 -17952.901,E2 -17952.901} C_VEL
LIN {X 0,Y 271.605,Z 471.579,A -85,B 0,C 180,E1 -17956.426,E2 -17956.426} C_VEL
LIN {X 0,Y 270.258,Z 465.558,A -85,B 0,C 180,E1 -17960.688,E2 -17960.688} C_VEL
LIN {X 0,Y 270.25,Z 465.447,A -85,B 0,C 180,E1 -17963.72,E2 -17963.72} C_VEL
LIN {X 0,Y 270.197,Z 465.455,A -85,B 0,C 180,E1 -17966.891,E2 -17966.891} C_VEL
LIN {X 0,Y 270.227,Z 465.448,A -85,B 0,C 180,E1 -17970.386,E2 -17970.386} C_VEL
LIN {X 0,Y 270.259,Z 465.434,A -85,B 0,C 180,E1 -17973.763,E2 -17973.763} C_VEL
LIN {X 0,Y 270.235,Z 465.436,A -85,B 0,C 180,E1 -17977.039,E2 -17977.039} C_VEL
LIN {X 0,Y 270.318,Z 465.437,A -85,B 0,C 180,E1 -17980.246,E2 -17980.246} C_VEL
LIN {X 0,Y 270.393,Z 465.424,A -85,B 0,C 180,E1 -17984.935,E2 -17984.935} C_VEL
LIN {X 0,Y 270.432,Z 465.425,A -85,B 0,C 180,E1 -17989.518,E2 -17989.518} C_VEL
LIN {X 0,Y 270.602,Z 465.401,A -85,B 0,C 180,E1 -17992.538,E2 -17992.538} C_VEL
LIN {X 0,Y 270.781,Z 465.374,A -85,B 0,C 180,E1 -17998.513,E2 -17998.513} C_VEL
LIN {X 0,Y 270.778,Z 465.374,A -85,B 0,C 180,E1 -18001.487,E2 -18001.487} C_VEL
LIN {X 0,Y 270.43,Z 465.396,A -85,B 0,C 180,E1 -18004.277,E2 -18004.277} C_VEL
LIN {X 0,Y 269.705,Z 465.503,A -85,B 0,C 180,E1 -18005.521,E2 -18005.521} C_VEL
LIN {X 0,Y 266.888,Z 465.866,A -85,B 0,C 180,E1 -18007.55,E2 -18007.55} C_VEL
LIN {X 0,Y 264.514,Z 466.145,A -85,B 0,C 180,E1 -18009.199,E2 -18009.199} C_VEL
LIN {X 0,Y 263.46,Z 466.263,A -85,B 0,C 180,E1 -18010.476,E2 -18010.476} C_VEL
LIN {X 0,Y 263.353,Z 466.276,A -85,B 0,C 180,E1 -18010.908,E2 -18010.908} C_VEL
LIN {X 0,Y 263.341,Z 466.3,A -85,B 0,C 180,E1 -18015.479,E2 -18015.479} C_VEL
LIN {X 0,Y 263.254,Z 466.318,A -85,B 0,C 180,E1 -18020.307,E2 -18020.307} C_VEL
LIN {X 0,Y 263.199,Z 466.321,A -85,B 0,C 180,E1 -18025.292,E2 -18025.292} C_VEL
LIN {X 0,Y 263.171,Z 466.326,A -85,B 0,C 180,E1 -18028.731,E2 -18028.731} C_VEL
LIN {X 0,Y 263.125,Z 466.336,A -85,B 0,C 180,E1 -18032.289,E2 -18032.289} C_VEL
LIN {X 0,Y 263.182,Z 466.325,A -85,B 0,C 180,E1 -18035.979,E2 -18035.979} C_VEL
LIN {X 0,Y 263.153,Z 466.332,A -85,B 0,C 180,E1 -18039.864,E2 -18039.864} C_VEL
LIN {X 0,Y 263.216,Z 466.498,A -85,B 0,C 180,E1 -18043.173,E2 -18043.173} C_VEL
LIN {X 0,Y 264.204,Z 471.954,A -85,B 0,C 180,E1 -18047.053,E2 -18047.053} C_VEL
LIN {X 0,Y 265.195,Z 477.033,A -85,B 0,C 180,E1 -18050.506,E2 -18050.506} C_VEL
LIN {X 0,Y 265.878,Z 480.705,A -85,B 0,C 180,E1 -18052.861,E2 -18052.861} C_VEL
LIN {X 0,Y 267.705,Z 488.998,A -85,B 0,C 180,E1 -18055.446,E2 -18055.446} C_VEL
LIN {X 0,Y 267.769,Z 492.101,A -85,B 0,C 180,E1 -18056.291,E2 -18056.291} C_VEL
LIN {X 0,Y 272.598,Z 507.927,A -85,B 0,C 180,E1 -18057.515,E2 -18057.515} C_VEL
LIN {X 0,Y 275.367,Z 521.563,A -85,B 0,C 180,E1 -18058.648,E2 -18058.648} C_VEL
LIN {X 0,Y 277.143,Z 535.379,A -85,B 0,C 180,E1 -18059.974,E2 -18059.974} C_VEL
LIN {X 0,Y 278.068,Z 547.199,A -85,B 0,C 180,E1 -18061.303,E2 -18061.303} C_VEL
LIN {X 0,Y 277.943,Z 552.355,A -85,B 0,C 180,E1 -18061.907,E2 -18061.907} C_VEL
LIN {X 0,Y 275.77,Z 563.854,A -85,B 0,C 180,E1 -18063.279,E2 -18063.279} C_VEL
LIN {X 0,Y 273.437,Z 574.879,A -85,B 0,C 180,E1 -18064.909,E2 -18064.909} C_VEL
LIN {X 0,Y 270.992,Z 584.88,A -85,B 0,C 180,E1 -18066.705,E2 -18066.705} C_VEL
LIN {X 0,Y 268.525,Z 594.812,A -85,B 0,C 180,E1 -18068.91,E2 -18068.91} C_VEL
LIN {X 0,Y 266.099,Z 604.27,A -85,B 0,C 180,E1 -18071.525,E2 -18071.525} C_VEL
LIN {X 0,Y 264.514,Z 610.899,A -85,B 0,C 180,E1 -18073.803,E2 -18073.803} C_VEL
LIN {X 0,Y 263.289,Z 616.393,A -85,B 0,C 180,E1 -18076.102,E2 -18076.102} C_VEL
LIN {X 0,Y 262.024,Z 622.143,A -85,B 0,C 180,E1 -18079.18,E2 -18079.18} C_VEL
LIN {X 0,Y 261.339,Z 626.317,A -85,B 0,C 180,E1 -18082.275,E2 -18082.275} C_VEL
LIN {X 0,Y 261.068,Z 629.039,A -85,B 0,C 180,E1 -18085.37,E2 -18085.37} C_VEL
LIN {X 0,Y 261.091,Z 630.387,A -85,B 0,C 180,E1 -18088.46,E2 -18088.46} C_VEL
LIN {X 0,Y 261.093,Z 630.378,A -85,B 0,C 180,E1 -18091.544,E2 -18091.544} C_VEL
LIN {X 0,Y 261.071,Z 629.013,A -85,B 0,C 180,E1 -18094.634,E2 -18094.634} C_VEL
LIN {X 0,Y 261.341,Z 626.276,A -85,B 0,C 180,E1 -18097.729,E2 -18097.729} C_VEL
LIN {X 0,Y 262.02,Z 622.091,A -85,B 0,C 180,E1 -18100.824,E2 -18100.824} C_VEL
LIN {X 0,Y 263.267,Z 616.327,A -85,B 0,C 180,E1 -18103.904,E2 -18103.904} C_VEL
LIN {X 0,Y 264.178,Z 613.192,A -85,B 0,C 180,E1 -18105.43,E2 -18105.43} C_VEL
LIN {X 0,Y 266.42,Z 607.916,A -85,B 0,C 180,E1 -18108.456,E2 -18108.456} C_VEL
LIN {X 0,Y 269.74,Z 601.169,A -85,B 0,C 180,E1 -18111.395,E2 -18111.395} C_VEL
LIN {X 0,Y 273.143,Z 594.009,A -85,B 0,C 180,E1 -18113.909,E2 -18113.909} C_VEL
LIN {X 0,Y 277.425,Z 585.435,A -85,B 0,C 180,E1 -18116.318,E2 -18116.318} C_VEL
LIN {X 0,Y 282.28,Z 575.301,A -85,B 0,C 180,E1 -18118.64,E2 -18118.64} C_VEL
LIN {X 0,Y 286.995,Z 565.109,A -85,B 0,C 180,E1 -18120.541,E2 -18120.541} C_VEL
LIN {X 0,Y 289.733,Z 558.814,A -85,B 0,C 180,E1 -18121.569,E2 -18121.569} C_VEL
LIN {X 0,Y 291.127,Z 552.242,A -85,B 0,C 180,E1 -18122.901,E2 -18122.901} C_VEL
LIN {X 0,Y 292.06,Z 542.695,A -85,B 0,C 180,E1 -18125.099,E2 -18125.099} C_VEL
LIN {X 0,Y 292.19,Z 535.665,A -85,B 0,C 180,E1 -18126.966,E2 -18126.966} C_VEL
LIN {X 0,Y 291.828,Z 532.359,A -85,B 0,C 180,E1 -18128.089,E2 -18128.089} C_VEL
LIN {X 0,Y 291.151,Z 529.354,A -85,B 0,C 180,E1 -18129.427,E2 -18129.427} C_VEL
LIN {X 0,Y 290.074,Z 526.313,A -85,B 0,C 180,E1 -18131.316,E2 -18131.316} C_VEL
LIN {X 0,Y 289.295,Z 524.166,A -85,B 0,C 180,E1 -18133.214,E2 -18133.214} C_VEL
LIN {X 0,Y 288.722,Z 523.056,A -85,B 0,C 180,E1 -18135.097,E2 -18135.097} C_VEL
LIN {X 0,Y 288.549,Z 522.598,A -85,B 0,C 180,E1 -18137.002,E2 -18137.002} C_VEL
LIN {X 0,Y 288.815,Z 522.799,A -85,B 0,C 180,E1 -18138.971,E2 -18138.971} C_VEL
LIN {X 0,Y 289.259,Z 524.309,A -85,B 0,C 180,E1 -18141.033,E2 -18141.033} C_VEL
LIN {X 0,Y 289.857,Z 527.141,A -85,B 0,C 180,E1 -18143.145,E2 -18143.145} C_VEL
LIN {X 0,Y 290.553,Z 532.315,A -85,B 0,C 180,E1 -18145.705,E2 -18145.705} C_VEL
LIN {X 0,Y 291.053,Z 537.344,A -85,B 0,C 180,E1 -18147.689,E2 -18147.689} C_VEL
LIN {X 0,Y 291.196,Z 544.254,A -85,B 0,C 180,E1 -18149.953,E2 -18149.953} C_VEL
LIN {X 0,Y 290.866,Z 548.902,A -85,B 0,C 180,E1 -18151.309,E2 -18151.309} C_VEL
LIN {X 0,Y 290.434,Z 550.625,A -85,B 0,C 180,E1 -18151.713,E2 -18151.713} C_VEL
LIN {X 0,Y 285.526,Z 560.907,A -85,B 0,C 180,E1 -18153.701,E2 -18153.701} C_VEL
LIN {X 0,Y 280.597,Z 570.416,A -85,B 0,C 180,E1 -18155.983,E2 -18155.983} C_VEL
LIN {X 0,Y 276.188,Z 578.27,A -85,B 0,C 180,E1 -18158.348,E2 -18158.348} C_VEL
LIN {X 0,Y 272.968,Z 583.833,A -85,B 0,C 180,E1 -18160.445,E2 -18160.445} C_VEL
LIN {X 0,Y 269.356,Z 589.733,A -85,B 0,C 180,E1 -18163.321,E2 -18163.321} C_VEL
LIN {X 0,Y 266.371,Z 594.082,A -85,B 0,C 180,E1 -18166.264,E2 -18166.264} C_VEL
LIN {X 0,Y 264.368,Z 596.923,A -85,B 0,C 180,E1 -18169.275,E2 -18169.275} C_VEL
LIN {X 0,Y 262.727,Z 598.313,A -85,B 0,C 180,E1 -18172.314,E2 -18172.314} C_VEL
LIN {X 0,Y 261.846,Z 598.227,A -85,B 0,C 180,E1 -18175.382,E2 -18175.382} C_VEL
LIN {X 0,Y 261.37,Z 596.67,A -85,B 0,C 180,E1 -18178.459,E2 -18178.459} C_VEL
LIN {X 0,Y 261.27,Z 595.297,A -85,B 0,C 180,E1 -18180,E2 -18180} C_VEL
LIN {X 0,Y 261.299,Z 592.51,A -85,B 0,C 180,E1 -18182.312,E2 -18182.312} C_VEL
LIN {X 0,Y 261.389,Z 588.717,A -85,B 0,C 180,E1 -18184.627,E2 -18184.627} C_VEL
LIN {X 0,Y 261.637,Z 583.875,A -85,B 0,C 180,E1 -18186.943,E2 -18186.943} C_VEL
LIN {X 0,Y 262.205,Z 576.74,A -85,B 0,C 180,E1 -18189.644,E2 -18189.644} C_VEL
LIN {X 0,Y 263.14,Z 567.788,A -85,B 0,C 180,E1 -18192.337,E2 -18192.337} C_VEL
LIN {X 0,Y 264.258,Z 558.277,A -85,B 0,C 180,E1 -18194.635,E2 -18194.635} C_VEL
LIN {X 0,Y 265.555,Z 547.67,A -85,B 0,C 180,E1 -18196.727,E2 -18196.727} C_VEL
LIN {X 0,Y 266.917,Z 536.098,A -85,B 0,C 180,E1 -18198.598,E2 -18198.598} C_VEL
LIN {X 0,Y 268.313,Z 522.998,A -85,B 0,C 180,E1 -18200.308,E2 -18200.308} C_VEL
LIN {X 0,Y 266.287,Z 509.869,A -85,B 0,C 180,E1 -18201.798,E2 -18201.798} C_VEL
LIN {X 0,Y 264.028,Z 495.954,A -85,B 0,C 180,E1 -18203.079,E2 -18203.079} C_VEL
LIN {X 0,Y 262.236,Z 484.916,A -85,B 0,C 180,E1 -18203.917,E2 -18203.917} C_VEL
LIN {X 0,Y 262.724,Z 479.904,A -85,B 0,C 180,E1 -18208.019,E2 -18208.019} C_VEL
LIN {X 0,Y 263.283,Z 474.855,A -85,B 0,C 180,E1 -18212.268,E2 -18212.268} C_VEL
LIN {X 0,Y 263.491,Z 470.628,A -85,B 0,C 180,E1 -18215.93,E2 -18215.93} C_VEL
LIN {X 0,Y 263.472,Z 467.205,A -85,B 0,C 180,E1 -18219.082,E2 -18219.082} C_VEL
LIN {X 0,Y 264.711,Z 473.529,A -85,B 0,C 180,E1 -18223.654,E2 -18223.654} C_VEL
LIN {X 0,Y 265.805,Z 479.543,A -85,B 0,C 180,E1 -18227.76,E2 -18227.76} C_VEL
LIN {X 0,Y 266.216,Z 482.919,A -85,B 0,C 180,E1 -18229.96,E2 -18229.96} C_VEL
LIN {X 0,Y 265.953,Z 487.274,A -85,B 0,C 180,E1 -18232.568,E2 -18232.568} C_VEL
LIN {X 0,Y 265.431,Z 493.161,A -85,B 0,C 180,E1 -18235.937,E2 -18235.937} C_VEL
LIN {X 0,Y 270.569,Z 507.777,A -85,B 0,C 180,E1 -18237.269,E2 -18237.269} C_VEL
LIN {X 0,Y 274.085,Z 520.406,A -85,B 0,C 180,E1 -18238.539,E2 -18238.539} C_VEL
LIN {X 0,Y 276.802,Z 533.952,A -85,B 0,C 180,E1 -18240.047,E2 -18240.047} C_VEL
LIN {X 0,Y 278.389,Z 546.88,A -85,B 0,C 180,E1 -18241.666,E2 -18241.666} C_VEL
LIN {X 0,Y 278.374,Z 549.46,A -85,B 0,C 180,E1 -18241.995,E2 -18241.995} C_VEL
LIN {X 0,Y 276.05,Z 561.856,A -85,B 0,C 180,E1 -18243.541,E2 -18243.541} C_VEL
LIN {X 0,Y 273.418,Z 573.34,A -85,B 0,C 180,E1 -18245.309,E2 -18245.309} C_VEL
LIN {X 0,Y 271.093,Z 582.863,A -85,B 0,C 180,E1 -18247.114,E2 -18247.114} C_VEL
LIN {X 0,Y 268.675,Z 592.397,A -85,B 0,C 180,E1 -18249.319,E2 -18249.319} C_VEL
LIN {X 0,Y 266.3,Z 601.175,A -85,B 0,C 180,E1 -18251.822,E2 -18251.822} C_VEL
LIN {X 0,Y 265.138,Z 606.874,A -85,B 0,C 180,E1 -18253.838,E2 -18253.838} C_VEL
LIN {X 0,Y 263.583,Z 612.333,A -85,B 0,C 180,E1 -18256.113,E2 -18256.113} C_VEL
LIN {X 0,Y 262.302,Z 618.041,A -85,B 0,C 180,E1 -18259.188,E2 -18259.188} C_VEL
LIN {X 0,Y 261.518,Z 622.19,A -85,B 0,C 180,E1 -18262.276,E2 -18262.276} C_VEL
LIN {X 0,Y 261.127,Z 624.908,A -85,B 0,C 180,E1 -18265.367,E2 -18265.367} C_VEL
LIN {X 0,Y 261.05,Z 626.271,A -85,B 0,C 180,E1 -18268.455,E2 -18268.455} C_VEL
LIN {X 0,Y 261.075,Z 626.454,A -85,B 0,C 180,E1 -18269.998,E2 -18269.998} C_VEL
LIN {X 0,Y 261.071,Z 625.819,A -85,B 0,C 180,E1 -18273.084,E2 -18273.084} C_VEL
LIN {X 0,Y 261.262,Z 623.839,A -85,B 0,C 180,E1 -18276.175,E2 -18276.175} C_VEL
LIN {X 0,Y 261.855,Z 620.469,A -85,B 0,C 180,E1 -18279.265,E2 -18279.265} C_VEL
LIN {X 0,Y 262.814,Z 615.611,A -85,B 0,C 180,E1 -18282.351,E2 -18282.351} C_VEL
LIN {X 0,Y 264.031,Z 610.904,A -85,B 0,C 180,E1 -18284.645,E2 -18284.645} C_VEL
LIN {X 0,Y 265.463,Z 605.182,A -85,B 0,C 180,E1 -18286.929,E2 -18286.929} C_VEL
LIN {X 0,Y 267.495,Z 596.947,A -85,B 0,C 180,E1 -18289.569,E2 -18289.569} C_VEL
LIN {X 0,Y 269.829,Z 588.356,A -85,B 0,C 180,E1 -18291.785,E2 -18291.785} C_VEL
LIN {X 0,Y 272.376,Z 577.945,A -85,B 0,C 180,E1 -18293.976,E2 -18293.976} C_VEL
LIN {X 0,Y 274.891,Z 567.445,A -85,B 0,C 180,E1 -18295.759,E2 -18295.759} C_VEL
LIN {X 0,Y 277.286,Z 555.69,A -85,B 0,C 180,E1 -18297.391,E2 -18297.391} C_VEL
LIN {X 0,Y 278.472,Z 548.301,A -85,B 0,C 180,E1 -18298.271,E2 -18298.271} C_VEL
LIN {X 0,Y 277.156,Z 536.183,A -85,B 0,C 180,E1 -18299.815,E2 -18299.815} C_VEL
LIN {X 0,Y 274.836,Z 523.431,A -85,B 0,C 180,E1 -18301.264,E2 -18301.264} C_VEL
LIN {X 0,Y 271.543,Z 510.782,A -85,B 0,C 180,E1 -18302.567,E2 -18302.567} C_VEL
LIN {X 0,Y 267.653,Z 499.308,A -85,B 0,C 180,E1 -18303.656,E2 -18303.656} C_VEL
LIN {X 0,Y 265.449,Z 493.079,A -85,B 0,C 180,E1 -18304.238,E2 -18304.238} C_VEL
LIN {X 0,Y 266.128,Z 485.928,A -85,B 0,C 180,E1 -18308.356,E2 -18308.356} C_VEL
LIN {X 0,Y 266.293,Z 483.125,A -85,B 0,C 180,E1 -18310.06,E2 -18310.06} C_VEL
LIN {X 0,Y 265.911,Z 479.732,A -85,B 0,C 180,E1 -18312.265,E2 -18312.265} C_VEL
LIN {X 0,Y 264.833,Z 473.702,A -85,B 0,C 180,E1 -18316.372,E2 -18316.372} C_VEL
LIN {X 0,Y 263.495,Z 467.737,A -85,B 0,C 180,E1 -18320.665,E2 -18320.665} C_VEL
LIN {X 0,Y 263.188,Z 466.325,A -85,B 0,C 180,E1 -18321.736,E2 -18321.736} C_VEL
LIN {X 0,Y 263.176,Z 466.321,A -85,B 0,C 180,E1 -18325.889,E2 -18325.889} C_VEL
LIN {X 0,Y 263.144,Z 466.323,A -85,B 0,C 180,E1 -18329.506,E2 -18329.506} C_VEL
LIN {X 0,Y 263.188,Z 466.314,A -85,B 0,C 180,E1 -18333.002,E2 -18333.002} C_VEL
LIN {X 0,Y 263.184,Z 466.322,A -85,B 0,C 180,E1 -18336.387,E2 -18336.387} C_VEL
LIN {X 0,Y 263.279,Z 466.309,A -85,B 0,C 180,E1 -18339.694,E2 -18339.694} C_VEL
LIN {X 0,Y 263.342,Z 466.304,A -85,B 0,C 180,E1 -18344.521,E2 -18344.521} C_VEL
LIN {X 0,Y 263.365,Z 466.303,A -85,B 0,C 180,E1 -18349.234,E2 -18349.234} C_VEL
LIN {X 0,Y 263.564,Z 466.276,A -85,B 0,C 180,E1 -18352.338,E2 -18352.338} C_VEL
LIN {X 0,Y 263.747,Z 466.25,A -85,B 0,C 180,E1 -18358.473,E2 -18358.473} C_VEL
LIN {X 0,Y 263.742,Z 466.25,A -85,B 0,C 180,E1 -18361.527,E2 -18361.527} C_VEL
LIN {X 0,Y 263.562,Z 466.281,A -85,B 0,C 180,E1 -18367.662,E2 -18367.662} C_VEL
LIN {X 0,Y 263.353,Z 466.276,A -85,B 0,C 180,E1 -18370.908,E2 -18370.908} C_VEL
LIN {X 0,Y 262.633,Z 466.378,A -85,B 0,C 180,E1 -18372.183,E2 -18372.183} C_VEL
LIN {X 0,Y 259.779,Z 466.751,A -85,B 0,C 180,E1 -18374.263,E2 -18374.263} C_VEL
LIN {X 0,Y 257.366,Z 467.037,A -85,B 0,C 180,E1 -18375.953,E2 -18375.953} C_VEL
LIN {X 0,Y 256.297,Z 467.158,A -85,B 0,C 180,E1 -18377.263,E2 -18377.263} C_VEL
LIN {X 0,Y 256.19,Z 467.171,A -85,B 0,C 180,E1 -18377.708,E2 -18377.708} C_VEL
LIN {X 0,Y 256.148,Z 467.203,A -85,B 0,C 180,E1 -18381.12,E2 -18381.12} C_VEL
LIN {X 0,Y 256.179,Z 467.195,A -85,B 0,C 180,E1 -18385.14,E2 -18385.14} C_VEL
LIN {X 0,Y 256.105,Z 467.21,A -85,B 0,C 180,E1 -18389.601,E2 -18389.601} C_VEL
LIN {X 0,Y 256.077,Z 467.211,A -85,B 0,C 180,E1 -18393.291,E2 -18393.291} C_VEL
LIN {X 0,Y 256.134,Z 467.205,A -85,B 0,C 180,E1 -18397.28,E2 -18397.28} C_VEL
LIN {X 0,Y 256.098,Z 467.207,A -85,B 0,C 180,E1 -18401.195,E2 -18401.195} C_VEL
LIN {X 0,Y 256.17,Z 467.328,A -85,B 0,C 180,E1 -18402.834,E2 -18402.834} C_VEL
LIN {X 0,Y 257.17,Z 472.892,A -85,B 0,C 180,E1 -18406.909,E2 -18406.909} C_VEL
LIN {X 0,Y 258.244,Z 478.414,A -85,B 0,C 180,E1 -18410.751,E2 -18410.751} C_VEL
LIN {X 0,Y 260.946,Z 489.812,A -85,B 0,C 180,E1 -18414.618,E2 -18414.618} C_VEL
LIN {X 0,Y 261.261,Z 492.314,A -85,B 0,C 180,E1 -18415.337,E2 -18415.337} C_VEL
LIN {X 0,Y 266.015,Z 507.466,A -85,B 0,C 180,E1 -18416.583,E2 -18416.583} C_VEL
LIN {X 0,Y 268.765,Z 520.331,A -85,B 0,C 180,E1 -18417.696,E2 -18417.696} C_VEL
LIN {X 0,Y 270.571,Z 533.641,A -85,B 0,C 180,E1 -18419,E2 -18419} C_VEL
LIN {X 0,Y 271.521,Z 545.521,A -85,B 0,C 180,E1 -18420.345,E2 -18420.345} C_VEL
LIN {X 0,Y 271.652,Z 552.322,A -85,B 0,C 180,E1 -18421.196,E2 -18421.196} C_VEL
LIN {X 0,Y 269.289,Z 564.52,A -85,B 0,C 180,E1 -18422.698,E2 -18422.698} C_VEL
LIN {X 0,Y 266.749,Z 575.899,A -85,B 0,C 180,E1 -18424.444,E2 -18424.444} C_VEL
LIN {X 0,Y 263.981,Z 586.607,A -85,B 0,C 180,E1 -18426.465,E2 -18426.465} C_VEL
LIN {X 0,Y 261.501,Z 596.243,A -85,B 0,C 180,E1 -18428.729,E2 -18428.729} C_VEL
LIN {X 0,Y 259.337,Z 604.22,A -85,B 0,C 180,E1 -18431.025,E2 -18431.025} C_VEL
LIN {X 0,Y 257.666,Z 610.847,A -85,B 0,C 180,E1 -18433.36,E2 -18433.36} C_VEL
LIN {X 0,Y 256.354,Z 616.34,A -85,B 0,C 180,E1 -18435.718,E2 -18435.718} C_VEL
LIN {X 0,Y 255.018,Z 622.089,A -85,B 0,C 180,E1 -18438.879,E2 -18438.879} C_VEL
LIN {X 0,Y 254.295,Z 626.262,A -85,B 0,C 180,E1 -18442.059,E2 -18442.059} C_VEL
LIN {X 0,Y 253.992,Z 628.984,A -85,B 0,C 180,E1 -18445.24,E2 -18445.24} C_VEL
LIN {X 0,Y 253.999,Z 630.331,A -85,B 0,C 180,E1 -18448.416,E2 -18448.416} C_VEL
LIN {X 0,Y 254,Z 630.322,A -85,B 0,C 180,E1 -18451.588,E2 -18451.588} C_VEL
LIN {X 0,Y 253.994,Z 628.957,A -85,B 0,C 180,E1 -18454.764,E2 -18454.764} C_VEL
LIN {X 0,Y 254.297,Z 626.22,A -85,B 0,C 180,E1 -18457.945,E2 -18457.945} C_VEL
LIN {X 0,Y 255.013,Z 622.035,A -85,B 0,C 180,E1 -18461.125,E2 -18461.125} C_VEL
LIN {X 0,Y 256.337,Z 616.271,A -85,B 0,C 180,E1 -18464.287,E2 -18464.287} C_VEL
LIN {X 0,Y 256.804,Z 614.567,A -85,B 0,C 180,E1 -18465.071,E2 -18465.071} C_VEL
LIN {X 0,Y 259.143,Z 609.59,A -85,B 0,C 180,E1 -18468.34,E2 -18468.34} C_VEL
LIN {X 0,Y 262.286,Z 603.798,A -85,B 0,C 180,E1 -18471.209,E2 -18471.209} C_VEL
LIN {X 0,Y 266.296,Z 596.267,A -85,B 0,C 180,E1 -18474.148,E2 -18474.148} C_VEL
LIN {X 0,Y 270.557,Z 588.333,A -85,B 0,C 180,E1 -18476.623,E2 -18476.623} C_VEL
LIN {X 0,Y 275.542,Z 578.94,A -85,B 0,C 180,E1 -18478.989,E2 -18478.989} C_VEL
LIN {X 0,Y 281.189,Z 567.846,A -85,B 0,C 180,E1 -18481.242,E2 -18481.242} C_VEL
LIN {X 0,Y 284.804,Z 559.972,A -85,B 0,C 180,E1 -18482.61,E2 -18482.61} C_VEL
LIN {X 0,Y 286.181,Z 553.925,A -85,B 0,C 180,E1 -18483.967,E2 -18483.967} C_VEL
LIN {X 0,Y 287.356,Z 545.074,A -85,B 0,C 180,E1 -18486.187,E2 -18486.187} C_VEL
LIN {X 0,Y 287.719,Z 540.024,A -85,B 0,C 180,E1 -18487.639,E2 -18487.639} C_VEL
LIN {X 0,Y 287.391,Z 536.309,A -85,B 0,C 180,E1 -18489.098,E2 -18489.098} C_VEL
LIN {X 0,Y 286.343,Z 532.276,A -85,B 0,C 180,E1 -18491.507,E2 -18491.507} C_VEL
LIN {X 0,Y 285.663,Z 530.126,A -85,B 0,C 180,E1 -18493.543,E2 -18493.543} C_VEL
LIN {X 0,Y 285.077,Z 528.906,A -85,B 0,C 180,E1 -18496.347,E2 -18496.347} C_VEL
LIN {X 0,Y 285.152,Z 528.857,A -85,B 0,C 180,E1 -18498.283,E2 -18498.283} C_VEL
LIN {X 0,Y 285.4,Z 529.79,A -85,B 0,C 180,E1 -18500.189,E2 -18500.189} C_VEL
LIN {X 0,Y 285.749,Z 531.715,A -85,B 0,C 180,E1 -18502.057,E2 -18502.057} C_VEL
LIN {X 0,Y 286.028,Z 535.214,A -85,B 0,C 180,E1 -18504.181,E2 -18504.181} C_VEL
LIN {X 0,Y 286.299,Z 540.413,A -85,B 0,C 180,E1 -18506.579,E2 -18506.579} C_VEL
LIN {X 0,Y 286.141,Z 546.86,A -85,B 0,C 180,E1 -18508.95,E2 -18508.95} C_VEL
LIN {X 0,Y 285.632,Z 551.848,A -85,B 0,C 180,E1 -18510.521,E2 -18510.521} C_VEL
LIN {X 0,Y 285.145,Z 553.458,A -85,B 0,C 180,E1 -18510.924,E2 -18510.924} C_VEL
LIN {X 0,Y 279.595,Z 564.007,A -85,B 0,C 180,E1 -18513.099,E2 -18513.099} C_VEL
LIN {X 0,Y 274.454,Z 572.96,A -85,B 0,C 180,E1 -18515.41,E2 -18515.41} C_VEL
LIN {X 0,Y 269.859,Z 580.389,A -85,B 0,C 180,E1 -18517.813,E2 -18517.813} C_VEL
LIN {X 0,Y 266.511,Z 585.598,A -85,B 0,C 180,E1 -18519.952,E2 -18519.952} C_VEL
LIN {X 0,Y 262.701,Z 591.146,A -85,B 0,C 180,E1 -18522.886,E2 -18522.886} C_VEL
LIN {X 0,Y 259.573,Z 595.204,A -85,B 0,C 180,E1 -18525.896,E2 -18525.896} C_VEL
LIN {X 0,Y 257.456,Z 597.714,A -85,B 0,C 180,E1 -18528.984,E2 -18528.984} C_VEL
LIN {X 0,Y 255.72,Z 598.858,A -85,B 0,C 180,E1 -18532.102,E2 -18532.102} C_VEL
LIN {X 0,Y 254.796,Z 598.556,A -85,B 0,C 180,E1 -18535.254,E2 -18535.254} C_VEL
LIN {X 0,Y 254.512,Z 597.843,A -85,B 0,C 180,E1 -18536.834,E2 -18536.834} C_VEL
LIN {X 0,Y 254.192,Z 595.242,A -85,B 0,C 180,E1 -18540,E2 -18540} C_VEL
LIN {X 0,Y 254.229,Z 592.268,A -85,B 0,C 180,E1 -18542.377,E2 -18542.377} C_VEL
LIN {X 0,Y 254.315,Z 587.353,A -85,B 0,C 180,E1 -18545.262,E2 -18545.262} C_VEL
LIN {X 0,Y 254.712,Z 581.392,A -85,B 0,C 180,E1 -18547.93,E2 -18547.93} C_VEL
LIN {X 0,Y 255.428,Z 573.49,A -85,B 0,C 180,E1 -18550.703,E2 -18550.703} C_VEL
LIN {X 0,Y 256.295,Z 565.146,A -85,B 0,C 180,E1 -18553.075,E2 -18553.075} C_VEL
LIN {X 0,Y 257.575,Z 555.063,A -85,B 0,C 180,E1 -18555.428,E2 -18555.428} C_VEL
LIN {X 0,Y 259.093,Z 543.035,A -85,B 0,C 180,E1 -18557.699,E2 -18557.699} C_VEL
LIN {X 0,Y 260.456,Z 531.219,A -85,B 0,C 180,E1 -18559.507,E2 -18559.507} C_VEL
LIN {X 0,Y 261.263,Z 523.732,A -85,B 0,C 180,E1 -18560.469,E2 -18560.469} C_VEL
LIN {X 0,Y 259.297,Z 510.802,A -85,B 0,C 180,E1 -18561.999,E2 -18561.999} C_VEL
LIN {X 0,Y 256.99,Z 496.511,A -85,B 0,C 180,E1 -18563.361,E2 -18563.361} C_VEL
LIN {X 0,Y 255.204,Z 485.084,A -85,B 0,C 180,E1 -18564.236,E2 -18564.236} C_VEL
LIN {X 0,Y 255.714,Z 480.106,A -85,B 0,C 180,E1 -18568.417,E2 -18568.417} C_VEL
LIN {X 0,Y 256.12,Z 476.267,A -85,B 0,C 180,E1 -18571.715,E2 -18571.715} C_VEL
LIN {X 0,Y 256.385,Z 472.364,A -85,B 0,C 180,E1 -18575.145,E2 -18575.145} C_VEL
LIN {X 0,Y 256.44,Z 468.685,A -85,B 0,C 180,E1 -18578.496,E2 -18578.496} C_VEL
LIN {X 0,Y 257.199,Z 471.969,A -85,B 0,C 180,E1 -18580.981,E2 -18580.981} C_VEL
LIN {X 0,Y 258.256,Z 477.555,A -85,B 0,C 180,E1 -18585.036,E2 -18585.036} C_VEL
LIN {X 0,Y 259.112,Z 482.374,A -85,B 0,C 180,E1 -18588.353,E2 -18588.353} C_VEL
LIN {X 0,Y 259.361,Z 485.599,A -85,B 0,C 180,E1 -18590.445,E2 -18590.445} C_VEL
LIN {X 0,Y 258.754,Z 492.538,A -85,B 0,C 180,E1 -18594.571,E2 -18594.571} C_VEL
LIN {X 0,Y 258.682,Z 493.141,A -85,B 0,C 180,E1 -18594.918,E2 -18594.918} C_VEL
LIN {X 0,Y 259.941,Z 496.641,A -85,B 0,C 180,E1 -18595.234,E2 -18595.234} C_VEL
LIN {X 0,Y 264.604,Z 509.82,A -85,B 0,C 180,E1 -18596.544,E2 -18596.544} C_VEL
LIN {X 0,Y 268.086,Z 522.918,A -85,B 0,C 180,E1 -18597.941,E2 -18597.941} C_VEL
LIN {X 0,Y 270.46,Z 535.332,A -85,B 0,C 180,E1 -18599.403,E2 -18599.403} C_VEL
LIN {X 0,Y 271.827,Z 547.124,A -85,B 0,C 180,E1 -18600.942,E2 -18600.942} C_VEL
LIN {X 0,Y 272.002,Z 549.863,A -85,B 0,C 180,E1 -18601.327,E2 -18601.327} C_VEL
LIN {X 0,Y 269.712,Z 561.903,A -85,B 0,C 180,E1 -18602.869,E2 -18602.869} C_VEL
LIN {X 0,Y 266.965,Z 573.39,A -85,B 0,C 180,E1 -18604.671,E2 -18604.671} C_VEL
LIN {X 0,Y 264.551,Z 582.915,A -85,B 0,C 180,E1 -18606.515,E2 -18606.515} C_VEL
LIN {X 0,Y 262.032,Z 592.451,A -85,B 0,C 180,E1 -18608.77,E2 -18608.77} C_VEL
LIN {X 0,Y 259.795,Z 600.356,A -85,B 0,C 180,E1 -18611.055,E2 -18611.055} C_VEL
LIN {X 0,Y 258.292,Z 606.929,A -85,B 0,C 180,E1 -18613.397,E2 -18613.397} C_VEL
LIN {X 0,Y 256.68,Z 612.388,A -85,B 0,C 180,E1 -18615.732,E2 -18615.732} C_VEL
LIN {X 0,Y 255.305,Z 618.097,A -85,B 0,C 180,E1 -18618.888,E2 -18618.888} C_VEL
LIN {X 0,Y 254.454,Z 622.246,A -85,B 0,C 180,E1 -18622.06,E2 -18622.06} C_VEL
LIN {X 0,Y 254.064,Z 624.964,A -85,B 0,C 180,E1 -18625.238,E2 -18625.238} C_VEL
LIN {X 0,Y 253.961,Z 626.327,A -85,B 0,C 180,E1 -18628.412,E2 -18628.412} C_VEL
LIN {X 0,Y 253.982,Z 626.51,A -85,B 0,C 180,E1 -18629.998,E2 -18629.998} C_VEL
LIN {X 0,Y 253.973,Z 625.874,A -85,B 0,C 180,E1 -18633.171,E2 -18633.171} C_VEL
LIN {X 0,Y 254.183,Z 623.894,A -85,B 0,C 180,E1 -18636.348,E2 -18636.348} C_VEL
LIN {X 0,Y 254.819,Z 620.524,A -85,B 0,C 180,E1 -18639.523,E2 -18639.523} C_VEL
LIN {X 0,Y 255.835,Z 615.665,A -85,B 0,C 180,E1 -18642.693,E2 -18642.693} C_VEL
LIN {X 0,Y 257.144,Z 610.957,A -85,B 0,C 180,E1 -18645.047,E2 -18645.047} C_VEL
LIN {X 0,Y 258.953,Z 604.06,A -85,B 0,C 180,E1 -18647.803,E2 -18647.803} C_VEL
LIN {X 0,Y 261.172,Z 595.662,A -85,B 0,C 180,E1 -18650.474,E2 -18650.474} C_VEL
LIN {X 0,Y 263.61,Z 586.801,A -85,B 0,C 180,E1 -18652.739,E2 -18652.739} C_VEL
LIN {X 0,Y 266.382,Z 576.071,A -85,B 0,C 180,E1 -18654.967,E2 -18654.967} C_VEL
LIN {X 0,Y 269.067,Z 565.181,A -85,B 0,C 180,E1 -18656.778,E2 -18656.778} C_VEL
LIN {X 0,Y 271.338,Z 554.166,A -85,B 0,C 180,E1 -18658.28,E2 -18658.28} C_VEL
LIN {X 0,Y 271.966,Z 550.574,A -85,B 0,C 180,E1 -18658.704,E2 -18658.704} C_VEL
LIN {X 0,Y 271.247,Z 540.878,A -85,B 0,C 180,E1 -18660.013,E2 -18660.013} C_VEL
LIN {X 0,Y 269.242,Z 528.156,A -85,B 0,C 180,E1 -18661.576,E2 -18661.576} C_VEL
LIN {X 0,Y 266.189,Z 515.214,A -85,B 0,C 180,E1 -18663.017,E2 -18663.017} C_VEL
LIN {X 0,Y 262.291,Z 502.974,A -85,B 0,C 180,E1 -18664.282,E2 -18664.282} C_VEL
LIN {X 0,Y 258.784,Z 493.467,A -85,B 0,C 180,E1 -18665.186,E2 -18665.186} C_VEL
LIN {X 0,Y 258.699,Z 493.152,A -85,B 0,C 180,E1 -18665.21,E2 -18665.21} C_VEL
LIN {X 0,Y 259.409,Z 485.859,A -85,B 0,C 180,E1 -18669.541,E2 -18669.541} C_VEL
LIN {X 0,Y 259.253,Z 482.679,A -85,B 0,C 180,E1 -18671.614,E2 -18671.614} C_VEL
LIN {X 0,Y 258.134,Z 476.261,A -85,B 0,C 180,E1 -18676.031,E2 -18676.031} C_VEL
LIN {X 0,Y 256.942,Z 470.888,A -85,B 0,C 180,E1 -18679.981,E2 -18679.981} C_VEL
LIN {X 0,Y 256.148,Z 467.198,A -85,B 0,C 180,E1 -18682.87,E2 -18682.87} C_VEL
LIN {X 0,Y 256.078,Z 467.211,A -85,B 0,C 180,E1 -18686.708,E2 -18686.708} C_VEL
LIN {X 0,Y 256.134,Z 467.207,A -85,B 0,C 180,E1 -18691.402,E2 -18691.402} C_VEL
LIN {X 0,Y 256.163,Z 467.202,A -85,B 0,C 180,E1 -18695.699,E2 -18695.699} C_VEL
LIN {X 0,Y 256.224,Z 467.18,A -85,B 0,C 180,E1 -18699.11,E2 -18699.11} C_VEL
LIN {X 0,Y 256.291,Z 467.185,A -85,B 0,C 180,E1 -18704.084,E2 -18704.084} C_VEL
LIN {X 0,Y 256.3,Z 467.18,A -85,B 0,C 180,E1 -18708.933,E2 -18708.933} C_VEL
LIN {X 0,Y 256.531,Z 467.151,A -85,B 0,C 180,E1 -18712.127,E2 -18712.127} C_VEL
LIN {X 0,Y 256.711,Z 467.126,A -85,B 0,C 180,E1 -18718.431,E2 -18718.431} C_VEL
LIN {X 0,Y 256.705,Z 467.124,A -85,B 0,C 180,E1 -18721.569,E2 -18721.569} C_VEL
LIN {X 0,Y 256.53,Z 467.154,A -85,B 0,C 180,E1 -18727.873,E2 -18727.873} C_VEL
LIN {X 0,Y 256.3,Z 467.154,A -85,B 0,C 180,E1 -18731.066,E2 -18731.066} C_VEL
LIN {X 0,Y 256.29,Z 467.17,A -85,B 0,C 180,E1 -18735.915,E2 -18735.915} C_VEL
LIN {X 0,Y 256.19,Z 467.171,A -85,B 0,C 180,E1 -18737.708,E2 -18737.708} C_VEL
LIN {X 0,Y 255.45,Z 467.276,A -85,B 0,C 180,E1 -18739.018,E2 -18739.018} C_VEL
LIN {X 0,Y 252.527,Z 467.654,A -85,B 0,C 180,E1 -18741.154,E2 -18741.154} C_VEL
LIN {X 0,Y 250.125,Z 467.951,A -85,B 0,C 180,E1 -18742.893,E2 -18742.893} C_VEL
LIN {X 0,Y 249.157,Z 468.074,A -85,B 0,C 180,E1 -18744.242,E2 -18744.242} C_VEL
LIN {X 0,Y 249.111,Z 468.074,A -85,B 0,C 180,E1 -18744.699,E2 -18744.699} C_VEL
LIN {X 0,Y 249.074,Z 468.083,A -85,B 0,C 180,E1 -18748.994,E2 -18748.994} C_VEL
LIN {X 0,Y 249.028,Z 468.093,A -85,B 0,C 180,E1 -18752.426,E2 -18752.426} C_VEL
LIN {X 0,Y 249.068,Z 468.082,A -85,B 0,C 180,E1 -18756.339,E2 -18756.339} C_VEL
LIN {X 0,Y 249.07,Z 468.086,A -85,B 0,C 180,E1 -18760.465,E2 -18760.465} C_VEL
LIN {X 0,Y 249.128,Z 468.289,A -85,B 0,C 180,E1 -18762.613,E2 -18762.613} C_VEL
LIN {X 0,Y 249.927,Z 472.808,A -85,B 0,C 180,E1 -18766.03,E2 -18766.03} C_VEL
LIN {X 0,Y 250.578,Z 476.198,A -85,B 0,C 180,E1 -18768.428,E2 -18768.428} C_VEL
LIN {X 0,Y 252.782,Z 485.217,A -85,B 0,C 180,E1 -18771.802,E2 -18771.802} C_VEL
LIN {X 0,Y 254.473,Z 492.3,A -85,B 0,C 180,E1 -18774.269,E2 -18774.269} C_VEL
LIN {X 0,Y 257.765,Z 501.29,A -85,B 0,C 180,E1 -18775.102,E2 -18775.102} C_VEL
LIN {X 0,Y 261.287,Z 514.31,A -85,B 0,C 180,E1 -18776.261,E2 -18776.261} C_VEL
LIN {X 0,Y 263.508,Z 527.617,A -85,B 0,C 180,E1 -18777.535,E2 -18777.535} C_VEL
LIN {X 0,Y 264.737,Z 539.999,A -85,B 0,C 180,E1 -18778.885,E2 -18778.885} C_VEL
LIN {X 0,Y 265.296,Z 552.288,A -85,B 0,C 180,E1 -18780.438,E2 -18780.438} C_VEL
LIN {X 0,Y 263.337,Z 562.684,A -85,B 0,C 180,E1 -18781.728,E2 -18781.728} C_VEL
LIN {X 0,Y 260.875,Z 573.714,A -85,B 0,C 180,E1 -18783.395,E2 -18783.395} C_VEL
LIN {X 0,Y 257.987,Z 584.788,A -85,B 0,C 180,E1 -18785.456,E2 -18785.456} C_VEL
LIN {X 0,Y 255.258,Z 594.715,A -85,B 0,C 180,E1 -18787.757,E2 -18787.757} C_VEL
LIN {X 0,Y 252.605,Z 604.169,A -85,B 0,C 180,E1 -18790.499,E2 -18790.499} C_VEL
LIN {X 0,Y 250.841,Z 610.795,A -85,B 0,C 180,E1 -18792.894,E2 -18792.894} C_VEL
LIN {X 0,Y 249.438,Z 616.287,A -85,B 0,C 180,E1 -18795.313,E2 -18795.313} C_VEL
LIN {X 0,Y 248.022,Z 622.034,A -85,B 0,C 180,E1 -18798.562,E2 -18798.562} C_VEL
LIN {X 0,Y 247.225,Z 626.207,A -85,B 0,C 180,E1 -18801.831,E2 -18801.831} C_VEL
LIN {X 0,Y 246.921,Z 628.929,A -85,B 0,C 180,E1 -18805.104,E2 -18805.104} C_VEL
LIN {X 0,Y 246.908,Z 630.276,A -85,B 0,C 180,E1 -18808.371,E2 -18808.371} C_VEL
LIN {X 0,Y 246.91,Z 630.267,A -85,B 0,C 180,E1 -18811.633,E2 -18811.633} C_VEL
LIN {X 0,Y 246.913,Z 628.844,A -85,B 0,C 180,E1 -18814.983,E2 -18814.983} C_VEL
LIN {X 0,Y 247.228,Z 626.164,A -85,B 0,C 180,E1 -18818.173,E2 -18818.173} C_VEL
LIN {X 0,Y 248.017,Z 621.979,A -85,B 0,C 180,E1 -18821.443,E2 -18821.443} C_VEL
LIN {X 0,Y 248.984,Z 617.825,A -85,B 0,C 180,E1 -18823.884,E2 -18823.884} C_VEL
LIN {X 0,Y 249.93,Z 614.731,A -85,B 0,C 180,E1 -18825.496,E2 -18825.496} C_VEL
LIN {X 0,Y 252.263,Z 610.32,A -85,B 0,C 180,E1 -18828.696,E2 -18828.696} C_VEL
LIN {X 0,Y 255.738,Z 604.599,A -85,B 0,C 180,E1 -18831.779,E2 -18831.779} C_VEL
LIN {X 0,Y 260.424,Z 596.491,A -85,B 0,C 180,E1 -18835.155,E2 -18835.155} C_VEL
LIN {X 0,Y 265.791,Z 587.52,A -85,B 0,C 180,E1 -18837.993,E2 -18837.993} C_VEL
LIN {X 0,Y 271.169,Z 578.201,A -85,B 0,C 180,E1 -18840.359,E2 -18840.359} C_VEL
LIN {X 0,Y 276.926,Z 567.759,A -85,B 0,C 180,E1 -18842.498,E2 -18842.498} C_VEL
LIN {X 0,Y 279.382,Z 563.048,A -85,B 0,C 180,E1 -18843.325,E2 -18843.325} C_VEL
LIN {X 0,Y 281.023,Z 557.365,A -85,B 0,C 180,E1 -18844.666,E2 -18844.666} C_VEL
LIN {X 0,Y 282.602,Z 549.003,A -85,B 0,C 180,E1 -18846.895,E2 -18846.895} C_VEL
LIN {X 0,Y 283.193,Z 544.306,A -85,B 0,C 180,E1 -18848.349,E2 -18848.349} C_VEL
LIN {X 0,Y 283.069,Z 541.249,A -85,B 0,C 180,E1 -18849.676,E2 -18849.676} C_VEL
LIN {X 0,Y 282.208,Z 537.441,A -85,B 0,C 180,E1 -18852.254,E2 -18852.254} C_VEL
LIN {X 0,Y 281.661,Z 535.734,A -85,B 0,C 180,E1 -18854.321,E2 -18854.321} C_VEL
LIN {X 0,Y 281.342,Z 534.94,A -85,B 0,C 180,E1 -18856.423,E2 -18856.423} C_VEL
LIN {X 0,Y 281.392,Z 534.967,A -85,B 0,C 180,E1 -18858.53,E2 -18858.53} C_VEL
LIN {X 0,Y 281.488,Z 535.377,A -85,B 0,C 180,E1 -18859.522,E2 -18859.522} C_VEL
LIN {X 0,Y 281.689,Z 537.77,A -85,B 0,C 180,E1 -18862.072,E2 -18862.072} C_VEL
LIN {X 0,Y 281.701,Z 541.032,A -85,B 0,C 180,E1 -18864.086,E2 -18864.086} C_VEL
LIN {X 0,Y 281.613,Z 544.844,A -85,B 0,C 180,E1 -18865.947,E2 -18865.947} C_VEL
LIN {X 0,Y 281.105,Z 550.833,A -85,B 0,C 180,E1 -18868.33,E2 -18868.33} C_VEL
LIN {X 0,Y 280.276,Z 555.451,A -85,B 0,C 180,E1 -18869.9,E2 -18869.9} C_VEL
LIN {X 0,Y 274.496,Z 565.741,A -85,B 0,C 180,E1 -18872.144,E2 -18872.144} C_VEL
LIN {X 0,Y 269.064,Z 574.403,A -85,B 0,C 180,E1 -18874.47,E2 -18874.47} C_VEL
LIN {X 0,Y 263.55,Z 582.49,A -85,B 0,C 180,E1 -18877.253,E2 -18877.253} C_VEL
LIN {X 0,Y 260.068,Z 587.384,A -85,B 0,C 180,E1 -18879.433,E2 -18879.433} C_VEL
LIN {X 0,Y 256.087,Z 592.565,A -85,B 0,C 180,E1 -18882.429,E2 -18882.429} C_VEL
LIN {X 0,Y 252.783,Z 596.25,A -85,B 0,C 180,E1 -18885.509,E2 -18885.509} C_VEL
LIN {X 0,Y 250.539,Z 598.504,A -85,B 0,C 180,E1 -18888.676,E2 -18888.676} C_VEL
LIN {X 0,Y 248.718,Z 599.399,A -85,B 0,C 180,E1 -18891.878,E2 -18891.878} C_VEL
LIN {X 0,Y 247.727,Z 598.805,A -85,B 0,C 180,E1 -18895.118,E2 -18895.118} C_VEL
LIN {X 0,Y 247.222,Z 596.753,A -85,B 0,C 180,E1 -18898.371,E2 -18898.371} C_VEL
LIN {X 0,Y 247.116,Z 595.174,A -85,B 0,C 180,E1 -18900,E2 -18900} C_VEL
LIN {X 0,Y 247.141,Z 592.003,A -85,B 0,C 180,E1 -18902.445,E2 -18902.445} C_VEL
LIN {X 0,Y 247.215,Z 587.859,A -85,B 0,C 180,E1 -18904.893,E2 -18904.893} C_VEL
LIN {X 0,Y 247.573,Z 581.879,A -85,B 0,C 180,E1 -18907.657,E2 -18907.657} C_VEL
LIN {X 0,Y 248.179,Z 575.091,A -85,B 0,C 180,E1 -18910.195,E2 -18910.195} C_VEL
LIN {X 0,Y 249.031,Z 567,A -85,B 0,C 180,E1 -18912.634,E2 -18912.634} C_VEL
LIN {X 0,Y 250.221,Z 557.203,A -85,B 0,C 180,E1 -18915.059,E2 -18915.059} C_VEL
LIN {X 0,Y 251.621,Z 546.348,A -85,B 0,C 180,E1 -18917.264,E2 -18917.264} C_VEL
LIN {X 0,Y 253.045,Z 534.621,A -85,B 0,C 180,E1 -18919.208,E2 -18919.208} C_VEL
LIN {X 0,Y 254.17,Z 524.185,A -85,B 0,C 180,E1 -18920.643,E2 -18920.643} C_VEL
LIN {X 0,Y 252.379,Z 512.301,A -85,B 0,C 180,E1 -18922.104,E2 -18922.104} C_VEL
LIN {X 0,Y 250.102,Z 498.061,A -85,B 0,C 180,E1 -18923.528,E2 -18923.528} C_VEL
LIN {X 0,Y 248.141,Z 485.263,A -85,B 0,C 180,E1 -18924.582,E2 -18924.582} C_VEL
LIN {X 0,Y 248.674,Z 480.311,A -85,B 0,C 180,E1 -18928.819,E2 -18928.819} C_VEL
LIN {X 0,Y 249.259,Z 475.177,A -85,B 0,C 180,E1 -18933.354,E2 -18933.354} C_VEL
LIN {X 0,Y 249.436,Z 470.355,A -85,B 0,C 180,E1 -18937.769,E2 -18937.769} C_VEL
LIN {X 0,Y 249.592,Z 470.699,A -85,B 0,C 180,E1 -18938.278,E2 -18938.278} C_VEL
LIN {X 0,Y 250.387,Z 473.797,A -85,B 0,C 180,E1 -18940.723,E2 -18940.723} C_VEL
LIN {X 0,Y 251.305,Z 478.697,A -85,B 0,C 180,E1 -18944.359,E2 -18944.359} C_VEL
LIN {X 0,Y 252.21,Z 483.878,A -85,B 0,C 180,E1 -18948.025,E2 -18948.025} C_VEL
LIN {X 0,Y 252.491,Z 487.137,A -85,B 0,C 180,E1 -18950.191,E2 -18950.191} C_VEL
LIN {X 0,Y 251.969,Z 493.1,A -85,B 0,C 180,E1 -18953.823,E2 -18953.823} C_VEL
LIN {X 0,Y 254.653,Z 500.311,A -85,B 0,C 180,E1 -18954.56,E2 -18954.56} C_VEL
LIN {X 0,Y 258.994,Z 513.17,A -85,B 0,C 180,E1 -18955.938,E2 -18955.938} C_VEL
LIN {X 0,Y 262.165,Z 525.875,A -85,B 0,C 180,E1 -18957.389,E2 -18957.389} C_VEL
LIN {X 0,Y 264.424,Z 539.023,A -85,B 0,C 180,E1 -18959.041,E2 -18959.041} C_VEL
LIN {X 0,Y 265.545,Z 550.287,A -85,B 0,C 180,E1 -18960.616,E2 -18960.616} C_VEL
LIN {X 0,Y 263.972,Z 559.406,A -85,B 0,C 180,E1 -18961.796,E2 -18961.796} C_VEL
LIN {X 0,Y 261.129,Z 571.339,A -85,B 0,C 180,E1 -18963.634,E2 -18963.634} C_VEL
LIN {X 0,Y 258.504,Z 581.215,A -85,B 0,C 180,E1 -18965.504,E2 -18965.504} C_VEL
LIN {X 0,Y 255.833,Z 591.041,A -85,B 0,C 180,E1 -18967.805,E2 -18967.805} C_VEL
LIN {X 0,Y 253.068,Z 600.41,A -85,B 0,C 180,E1 -18970.532,E2 -18970.532} C_VEL
LIN {X 0,Y 251.444,Z 606.985,A -85,B 0,C 180,E1 -18972.932,E2 -18972.932} C_VEL
LIN {X 0,Y 249.795,Z 612.444,A -85,B 0,C 180,E1 -18975.33,E2 -18975.33} C_VEL
LIN {X 0,Y 248.301,Z 618.154,A -85,B 0,C 180,E1 -18978.57,E2 -18978.57} C_VEL
LIN {X 0,Y 247.403,Z 622.302,A -85,B 0,C 180,E1 -18981.832,E2 -18981.832} C_VEL
LIN {X 0,Y 246.972,Z 625.02,A -85,B 0,C 180,E1 -18985.101,E2 -18985.101} C_VEL
LIN {X 0,Y 246.874,Z 626.383,A -85,B 0,C 180,E1 -18988.367,E2 -18988.367} C_VEL
LIN {X 0,Y 246.893,Z 626.565,A -85,B 0,C 180,E1 -18989.998,E2 -18989.998} C_VEL
LIN {X 0,Y 246.879,Z 625.93,A -85,B 0,C 180,E1 -18993.262,E2 -18993.262} C_VEL
LIN {X 0,Y 247.121,Z 623.949,A -85,B 0,C 180,E1 -18996.53,E2 -18996.53} C_VEL
LIN {X 0,Y 247.805,Z 620.578,A -85,B 0,C 180,E1 -18999.795,E2 -18999.795} C_VEL
LIN {X 0,Y 248.87,Z 615.719,A -85,B 0,C 180,E1 -19003.055,E2 -19003.055} C_VEL
LIN {X 0,Y 250.839,Z 609.224,A -85,B 0,C 180,E1 -19006.269,E2 -19006.269} C_VEL
LIN {X 0,Y 252.59,Z 602.421,A -85,B 0,C 180,E1 -19008.913,E2 -19008.913} C_VEL
LIN {X 0,Y 254.895,Z 594.377,A -85,B 0,C 180,E1 -19011.426,E2 -19011.426} C_VEL
LIN {X 0,Y 257.493,Z 585.241,A -85,B 0,C 180,E1 -19013.738,E2 -19013.738} C_VEL
LIN {X 0,Y 260.248,Z 575.125,A -85,B 0,C 180,E1 -19015.812,E2 -19015.812} C_VEL
LIN {X 0,Y 262.998,Z 563.986,A -85,B 0,C 180,E1 -19017.662,E2 -19017.662} C_VEL
LIN {X 0,Y 265.553,Z 551.694,A -85,B 0,C 180,E1 -19019.312,E2 -19019.312} C_VEL
LIN {X 0,Y 264.704,Z 540.905,A -85,B 0,C 180,E1 -19020.834,E2 -19020.834} C_VEL
LIN {X 0,Y 262.912,Z 529.407,A -85,B 0,C 180,E1 -19022.316,E2 -19022.316} C_VEL
LIN {X 0,Y 260.17,Z 517.39,A -85,B 0,C 180,E1 -19023.731,E2 -19023.731} C_VEL
LIN {X 0,Y 256.503,Z 505.488,A -85,B 0,C 180,E1 -19025.037,E2 -19025.037} C_VEL
LIN {X 0,Y 252.006,Z 493.072,A -85,B 0,C 180,E1 -19026.345,E2 -19026.345} C_VEL
LIN {X 0,Y 252.546,Z 487.427,A -85,B 0,C 180,E1 -19029.793,E2 -19029.793} C_VEL
LIN {X 0,Y 252.333,Z 484.153,A -85,B 0,C 180,E1 -19031.944,E2 -19031.944} C_VEL
LIN {X 0,Y 251.442,Z 478.85,A -85,B 0,C 180,E1 -19035.671,E2 -19035.671} C_VEL
LIN {X 0,Y 250.437,Z 474.074,A -85,B 0,C 180,E1 -19039.258,E2 -19039.258} C_VEL
LIN {X 0,Y 249.459,Z 469.606,A -85,B 0,C 180,E1 -19042.719,E2 -19042.719} C_VEL
LIN {X 0,Y 249.065,Z 468.088,A -85,B 0,C 180,E1 -19044.01,E2 -19044.01} C_VEL
LIN {X 0,Y 249.032,Z 468.087,A -85,B 0,C 180,E1 -19047.843,E2 -19047.843} C_VEL
LIN {X 0,Y 249.092,Z 468.085,A -85,B 0,C 180,E1 -19051.338,E2 -19051.338} C_VEL
LIN {X 0,Y 249.146,Z 468.074,A -85,B 0,C 180,E1 -19054.968,E2 -19054.968} C_VEL
LIN {X 0,Y 249.122,Z 468.06,A -85,B 0,C 180,E1 -19058.579,E2 -19058.579} C_VEL
LIN {X 0,Y 249.233,Z 468.066,A -85,B 0,C 180,E1 -19063.621,E2 -19063.621} C_VEL
LIN {X 0,Y 249.244,Z 468.058,A -85,B 0,C 180,E1 -19068.616,E2 -19068.616} C_VEL
LIN {X 0,Y 249.475,Z 468.029,A -85,B 0,C 180,E1 -19071.902,E2 -19071.902} C_VEL
LIN {X 0,Y 249.454,Z 468.037,A -85,B 0,C 180,E1 -19076.77,E2 -19076.77} C_VEL
LIN {X 0,Y 249.726,Z 468.004,A -85,B 0,C 180,E1 -19080,E2 -19080} C_VEL
LIN {X 0,Y 249.427,Z 468.01,A -85,B 0,C 180,E1 -19083.23,E2 -19083.23} C_VEL
LIN {X 0,Y 249.474,Z 468.031,A -85,B 0,C 180,E1 -19088.097,E2 -19088.097} C_VEL
LIN {X 0,Y 249.244,Z 468.035,A -85,B 0,C 180,E1 -19091.384,E2 -19091.384} C_VEL
LIN {X 0,Y 249.232,Z 468.042,A -85,B 0,C 180,E1 -19096.379,E2 -19096.379} C_VEL
LIN {X 0,Y 249.078,Z 468.082,A -85,B 0,C 180,E1 -19101.519,E2 -19101.519} C_VEL
LIN {X 0,Y 249.111,Z 468.074,A -85,B 0,C 180,E1 -19104.699,E2 -19104.699} C_VEL
LIN {X 0,Y 248.851,Z 468.11,A -85,B 0,C 180,E1 -19105.601,E2 -19105.601} C_VEL
LIN {X 0,Y 247.525,Z 468.28,A -85,B 0,C 180,E1 -19106.934,E2 -19106.934} C_VEL
LIN {X 0,Y 243.118,Z 468.828,A -85,B 0,C 180,E1 -19110.039,E2 -19110.039} C_VEL
LIN {X 0,Y 242.047,Z 468.957,A -85,B 0,C 180,E1 -19111.431,E2 -19111.431} C_VEL
LIN {X 0,Y 241.964,Z 468.968,A -85,B 0,C 180,E1 -19111.903,E2 -19111.903} C_VEL
LIN {X 0,Y 242.021,Z 468.963,A -85,B 0,C 180,E1 -19115.606,E2 -19115.606} C_VEL
LIN {X 0,Y 242.001,Z 468.965,A -85,B 0,C 180,E1 -19119.71,E2 -19119.71} C_VEL
LIN {X 0,Y 242.07,Z 468.957,A -85,B 0,C 180,E1 -19122.174,E2 -19122.174} C_VEL
LIN {X 0,Y 242.84,Z 473.345,A -85,B 0,C 180,E1 -19125.576,E2 -19125.576} C_VEL
LIN {X 0,Y 244.785,Z 481.344,A -85,B 0,C 180,E1 -19128.907,E2 -19128.907} C_VEL
LIN {X 0,Y 246.854,Z 489.844,A -85,B 0,C 180,E1 -19132.191,E2 -19132.191} C_VEL
LIN {X 0,Y 247.35,Z 492.225,A -85,B 0,C 180,E1 -19133.066,E2 -19133.066} C_VEL
LIN {X 0,Y 250.624,Z 499.104,A -85,B 0,C 180,E1 -19133.869,E2 -19133.869} C_VEL
LIN {X 0,Y 254.404,Z 512.065,A -85,B 0,C 180,E1 -19135.087,E2 -19135.087} C_VEL
LIN {X 0,Y 256.838,Z 524.835,A -85,B 0,C 180,E1 -19136.352,E2 -19136.352} C_VEL
LIN {X 0,Y 258.241,Z 537.562,A -85,B 0,C 180,E1 -19137.751,E2 -19137.751} C_VEL
LIN {X 0,Y 258.866,Z 550.609,A -85,B 0,C 180,E1 -19139.402,E2 -19139.402} C_VEL
LIN {X 0,Y 258.688,Z 555.392,A -85,B 0,C 180,E1 -19140.055,E2 -19140.055} C_VEL
LIN {X 0,Y 256.103,Z 567.206,A -85,B 0,C 180,E1 -19141.647,E2 -19141.647} C_VEL
LIN {X 0,Y 253.143,Z 578.989,A -85,B 0,C 180,E1 -19143.63,E2 -19143.63} C_VEL
LIN {X 0,Y 250.036,Z 589.942,A -85,B 0,C 180,E1 -19145.95,E2 -19145.95} C_VEL
LIN {X 0,Y 247.397,Z 598.968,A -85,B 0,C 180,E1 -19148.33,E2 -19148.33} C_VEL
LIN {X 0,Y 245.116,Z 606.694,A -85,B 0,C 180,E1 -19150.837,E2 -19150.837} C_VEL
LIN {X 0,Y 243.467,Z 612.717,A -85,B 0,C 180,E1 -19153.224,E2 -19153.224} C_VEL
LIN {X 0,Y 242.08,Z 617.842,A -85,B 0,C 180,E1 -19155.716,E2 -19155.716} C_VEL
LIN {X 0,Y 241.02,Z 621.98,A -85,B 0,C 180,E1 -19158.225,E2 -19158.225} C_VEL
LIN {X 0,Y 240.177,Z 626.152,A -85,B 0,C 180,E1 -19161.589,E2 -19161.589} C_VEL
LIN {X 0,Y 239.837,Z 628.951,A -85,B 0,C 180,E1 -19165.075,E2 -19165.075} C_VEL
LIN {X 0,Y 239.819,Z 630.22,A -85,B 0,C 180,E1 -19168.323,E2 -19168.323} C_VEL
LIN {X 0,Y 239.825,Z 630.385,A -85,B 0,C 180,E1 -19170.002,E2 -19170.002} C_VEL
LIN {X 0,Y 239.821,Z 630.211,A -85,B 0,C 180,E1 -19171.681,E2 -19171.681} C_VEL
LIN {X 0,Y 239.841,Z 628.845,A -85,B 0,C 180,E1 -19175.045,E2 -19175.045} C_VEL
LIN {X 0,Y 240.179,Z 626.108,A -85,B 0,C 180,E1 -19178.415,E2 -19178.415} C_VEL
LIN {X 0,Y 241.014,Z 621.923,A -85,B 0,C 180,E1 -19181.78,E2 -19181.78} C_VEL
LIN {X 0,Y 242.069,Z 617.769,A -85,B 0,C 180,E1 -19184.289,E2 -19184.289} C_VEL
LIN {X 0,Y 243.07,Z 614.958,A -85,B 0,C 180,E1 -19185.945,E2 -19185.945} C_VEL
LIN {X 0,Y 245.437,Z 611.015,A -85,B 0,C 180,E1 -19189.101,E2 -19189.101} C_VEL
LIN {X 0,Y 249.196,Z 605.412,A -85,B 0,C 180,E1 -19192.381,E2 -19192.381} C_VEL
LIN {X 0,Y 253.593,Z 598.653,A -85,B 0,C 180,E1 -19195.442,E2 -19195.442} C_VEL
LIN {X 0,Y 258.239,Z 591.519,A -85,B 0,C 180,E1 -19198.001,E2 -19198.001} C_VEL
LIN {X 0,Y 264.461,Z 581.776,A -85,B 0,C 180,E1 -19200.77,E2 -19200.77} C_VEL
LIN {X 0,Y 270.626,Z 571.654,A -85,B 0,C 180,E1 -19203.051,E2 -19203.051} C_VEL
LIN {X 0,Y 274.401,Z 565.037,A -85,B 0,C 180,E1 -19204.298,E2 -19204.298} C_VEL
LIN {X 0,Y 276.334,Z 559.165,A -85,B 0,C 180,E1 -19205.802,E2 -19205.802} C_VEL
LIN {X 0,Y 278.19,Z 551.441,A -85,B 0,C 180,E1 -19208.07,E2 -19208.07} C_VEL
LIN {X 0,Y 278.607,Z 548.526,A -85,B 0,C 180,E1 -19209.099,E2 -19209.099} C_VEL
LIN {X 0,Y 278.658,Z 546.779,A -85,B 0,C 180,E1 -19209.895,E2 -19209.895} C_VEL
LIN {X 0,Y 278.227,Z 543.874,A -85,B 0,C 180,E1 -19211.828,E2 -19211.828} C_VEL
LIN {X 0,Y 277.926,Z 542.571,A -85,B 0,C 180,E1 -19213.061,E2 -19213.061} C_VEL
LIN {X 0,Y 277.495,Z 541.226,A -85,B 0,C 180,E1 -19215.167,E2 -19215.167} C_VEL
LIN {X 0,Y 277.361,Z 540.724,A -85,B 0,C 180,E1 -19217.295,E2 -19217.295} C_VEL
LIN {X 0,Y 277.438,Z 541.229,A -85,B 0,C 180,E1 -19219.462,E2 -19219.462} C_VEL
LIN {X 0,Y 277.425,Z 543.232,A -85,B 0,C 180,E1 -19221.753,E2 -19221.753} C_VEL
LIN {X 0,Y 277.072,Z 547.263,A -85,B 0,C 180,E1 -19224.31,E2 -19224.31} C_VEL
LIN {X 0,Y 276.501,Z 551.967,A -85,B 0,C 180,E1 -19226.559,E2 -19226.559} C_VEL
LIN {X 0,Y 275.523,Z 557.091,A -85,B 0,C 180,E1 -19228.582,E2 -19228.582} C_VEL
LIN {X 0,Y 274.806,Z 559.159,A -85,B 0,C 180,E1 -19229.237,E2 -19229.237} C_VEL
LIN {X 0,Y 267.789,Z 570.147,A -85,B 0,C 180,E1 -19231.81,E2 -19231.81} C_VEL
LIN {X 0,Y 261.546,Z 579.006,A -85,B 0,C 180,E1 -19234.537,E2 -19234.537} C_VEL
LIN {X 0,Y 255.98,Z 586.212,A -85,B 0,C 180,E1 -19237.395,E2 -19237.395} C_VEL
LIN {X 0,Y 251.442,Z 591.72,A -85,B 0,C 180,E1 -19240.403,E2 -19240.403} C_VEL
LIN {X 0,Y 247.665,Z 595.783,A -85,B 0,C 180,E1 -19243.515,E2 -19243.515} C_VEL
LIN {X 0,Y 246.001,Z 597.324,A -85,B 0,C 180,E1 -19245.101,E2 -19245.101} C_VEL
LIN {X 0,Y 243.617,Z 599.269,A -85,B 0,C 180,E1 -19248.35,E2 -19248.35} C_VEL
LIN {X 0,Y 241.704,Z 599.856,A -85,B 0,C 180,E1 -19251.641,E2 -19251.641} C_VEL
LIN {X 0,Y 240.662,Z 599.022,A -85,B 0,C 180,E1 -19254.974,E2 -19254.974} C_VEL
LIN {X 0,Y 240.151,Z 596.745,A -85,B 0,C 180,E1 -19258.323,E2 -19258.323} C_VEL
LIN {X 0,Y 240.05,Z 592.886,A -85,B 0,C 180,E1 -19261.678,E2 -19261.678} C_VEL
LIN {X 0,Y 240.102,Z 588.919,A -85,B 0,C 180,E1 -19264.197,E2 -19264.197} C_VEL
LIN {X 0,Y 240.35,Z 583.864,A -85,B 0,C 180,E1 -19266.717,E2 -19266.717} C_VEL
LIN {X 0,Y 240.934,Z 576.475,A -85,B 0,C 180,E1 -19269.656,E2 -19269.656} C_VEL
LIN {X 0,Y 241.762,Z 568.7,A -85,B 0,C 180,E1 -19272.167,E2 -19272.167} C_VEL
LIN {X 0,Y 242.848,Z 559.256,A -85,B 0,C 180,E1 -19274.669,E2 -19274.669} C_VEL
LIN {X 0,Y 244.163,Z 548.779,A -85,B 0,C 180,E1 -19276.944,E2 -19276.944} C_VEL
LIN {X 0,Y 245.333,Z 539.587,A -85,B 0,C 180,E1 -19278.609,E2 -19278.609} C_VEL
LIN {X 0,Y 246.846,Z 527.682,A -85,B 0,C 180,E1 -19280.412,E2 -19280.412} C_VEL
LIN {X 0,Y 247.05,Z 524.532,A -85,B 0,C 180,E1 -19280.83,E2 -19280.83} C_VEL
LIN {X 0,Y 245.157,Z 512.008,A -85,B 0,C 180,E1 -19282.415,E2 -19282.415} C_VEL
LIN {X 0,Y 242.917,Z 497.565,A -85,B 0,C 180,E1 -19283.894,E2 -19283.894} C_VEL
LIN {X 0,Y 241.106,Z 485.419,A -85,B 0,C 180,E1 -19284.908,E2 -19284.908} C_VEL
LIN {X 0,Y 241.639,Z 480.503,A -85,B 0,C 180,E1 -19289.241,E2 -19289.241} C_VEL
LIN {X 0,Y 242.22,Z 475.85,A -85,B 0,C 180,E1 -19293.455,E2 -19293.455} C_VEL
LIN {X 0,Y 242.396,Z 471.862,A -85,B 0,C 180,E1 -19297.259,E2 -19297.259} C_VEL
LIN {X 0,Y 243.346,Z 474.427,A -85,B 0,C 180,E1 -19299.448,E2 -19299.448} C_VEL
LIN {X 0,Y 244.448,Z 480.406,A -85,B 0,C 180,E1 -19304.045,E2 -19304.045} C_VEL
LIN {X 0,Y 245.435,Z 486.032,A -85,B 0,C 180,E1 -19308.117,E2 -19308.117} C_VEL
LIN {X 0,Y 245.597,Z 489.75,A -85,B 0,C 180,E1 -19310.591,E2 -19310.591} C_VEL
LIN {X 0,Y 245.328,Z 493.365,A -85,B 0,C 180,E1 -19312.712,E2 -19312.712} C_VEL
LIN {X 0,Y 250.829,Z 508.233,A -85,B 0,C 180,E1 -19314.347,E2 -19314.347} C_VEL
LIN {X 0,Y 254.546,Z 520.958,A -85,B 0,C 180,E1 -19315.846,E2 -19315.846} C_VEL
LIN {X 0,Y 257.015,Z 533.06,A -85,B 0,C 180,E1 -19317.364,E2 -19317.364} C_VEL
LIN {X 0,Y 258.54,Z 544.249,A -85,B 0,C 180,E1 -19318.901,E2 -19318.901} C_VEL
LIN {X 0,Y 259.14,Z 552.339,A -85,B 0,C 180,E1 -19320.108,E2 -19320.108} C_VEL
LIN {X 0,Y 256.537,Z 564.529,A -85,B 0,C 180,E1 -19321.796,E2 -19321.796} C_VEL
LIN {X 0,Y 253.612,Z 575.579,A -85,B 0,C 180,E1 -19323.678,E2 -19323.678} C_VEL
LIN {X 0,Y 250.605,Z 586.414,A -85,B 0,C 180,E1 -19326.004,E2 -19326.004} C_VEL
LIN {X 0,Y 247.935,Z 595.359,A -85,B 0,C 180,E1 -19328.375,E2 -19328.375} C_VEL
LIN {X 0,Y 245.398,Z 603.721,A -85,B 0,C 180,E1 -19331.13,E2 -19331.13} C_VEL
LIN {X 0,Y 244.07,Z 609.005,A -85,B 0,C 180,E1 -19333.263,E2 -19333.263} C_VEL
LIN {X 0,Y 241.999,Z 615.56,A -85,B 0,C 180,E1 -19336.564,E2 -19336.564} C_VEL
LIN {X 0,Y 240.779,Z 620.47,A -85,B 0,C 180,E1 -19339.912,E2 -19339.912} C_VEL
LIN {X 0,Y 240.058,Z 623.89,A -85,B 0,C 180,E1 -19343.273,E2 -19343.273} C_VEL
LIN {X 0,Y 239.791,Z 625.924,A -85,B 0,C 180,E1 -19346.637,E2 -19346.637} C_VEL
LIN {X 0,Y 239.805,Z 626.621,A -85,B 0,C 180,E1 -19349.998,E2 -19349.998} C_VEL
LIN {X 0,Y 239.788,Z 625.985,A -85,B 0,C 180,E1 -19353.358,E2 -19353.358} C_VEL
LIN {X 0,Y 240.056,Z 624.004,A -85,B 0,C 180,E1 -19356.723,E2 -19356.723} C_VEL
LIN {X 0,Y 240.769,Z 620.633,A -85,B 0,C 180,E1 -19360.084,E2 -19360.084} C_VEL
LIN {X 0,Y 241.921,Z 615.772,A -85,B 0,C 180,E1 -19363.436,E2 -19363.436} C_VEL
LIN {X 0,Y 244.006,Z 609.276,A -85,B 0,C 180,E1 -19366.737,E2 -19366.737} C_VEL
LIN {X 0,Y 245.864,Z 602.421,A -85,B 0,C 180,E1 -19369.471,E2 -19369.471} C_VEL
LIN {X 0,Y 248.289,Z 594.426,A -85,B 0,C 180,E1 -19372.025,E2 -19372.025} C_VEL
LIN {X 0,Y 250.986,Z 585.288,A -85,B 0,C 180,E1 -19374.392,E2 -19374.392} C_VEL
LIN {X 0,Y 253.868,Z 575.168,A -85,B 0,C 180,E1 -19376.51,E2 -19376.51} C_VEL
LIN {X 0,Y 256.669,Z 564.274,A -85,B 0,C 180,E1 -19378.361,E2 -19378.361} C_VEL
LIN {X 0,Y 259.147,Z 552.34,A -85,B 0,C 180,E1 -19380.021,E2 -19380.021} C_VEL
LIN {X 0,Y 258.353,Z 541.999,A -85,B 0,C 180,E1 -19381.551,E2 -19381.551} C_VEL
LIN {X 0,Y 256.402,Z 529.423,A -85,B 0,C 180,E1 -19383.241,E2 -19383.241} C_VEL
LIN {X 0,Y 253.664,Z 517.486,A -85,B 0,C 180,E1 -19384.71,E2 -19384.71} C_VEL
LIN {X 0,Y 250.086,Z 506.118,A -85,B 0,C 180,E1 -19386.036,E2 -19386.036} C_VEL
LIN {X 0,Y 245.867,Z 495.141,A -85,B 0,C 180,E1 -19387.269,E2 -19387.269} C_VEL
LIN {X 0,Y 245.281,Z 493.096,A -85,B 0,C 180,E1 -19387.491,E2 -19387.491} C_VEL
LIN {X 0,Y 245.701,Z 488.851,A -85,B 0,C 180,E1 -19390.149,E2 -19390.149} C_VEL
LIN {X 0,Y 245.314,Z 484.893,A -85,B 0,C 180,E1 -19392.826,E2 -19392.826} C_VEL
LIN {X 0,Y 244.487,Z 480.054,A -85,B 0,C 180,E1 -19396.377,E2 -19396.377} C_VEL
LIN {X 0,Y 243.324,Z 474.686,A -85,B 0,C 180,E1 -19400.548,E2 -19400.548} C_VEL
LIN {X 0,Y 242.28,Z 470.088,A -85,B 0,C 180,E1 -19404.309,E2 -19404.309} C_VEL
LIN {X 0,Y 242.011,Z 468.957,A -85,B 0,C 180,E1 -19405.382,E2 -19405.382} C_VEL
LIN {X 0,Y 242.023,Z 468.96,A -85,B 0,C 180,E1 -19410.419,E2 -19410.419} C_VEL
LIN {X 0,Y 242.059,Z 468.947,A -85,B 0,C 180,E1 -19414.182,E2 -19414.182} C_VEL
LIN {X 0,Y 242.076,Z 468.937,A -85,B 0,C 180,E1 -19418.277,E2 -19418.277} C_VEL
LIN {X 0,Y 242.154,Z 468.946,A -85,B 0,C 180,E1 -19423.277,E2 -19423.277} C_VEL
LIN {X 0,Y 242.178,Z 468.937,A -85,B 0,C 180,E1 -19428.279,E2 -19428.279} C_VEL
LIN {X 0,Y 242.426,Z 468.906,A -85,B 0,C 180,E1 -19431.665,E2 -19431.665} C_VEL
LIN {X 0,Y 242.256,Z 468.927,A -85,B 0,C 180,E1 -19435.007,E2 -19435.007} C_VEL
LIN {X 0,Y 242.635,Z 468.879,A -85,B 0,C 180,E1 -19438.34,E2 -19438.34} C_VEL
LIN {X 0,Y 242.627,Z 468.874,A -85,B 0,C 180,E1 -19441.66,E2 -19441.66} C_VEL
LIN {X 0,Y 242.424,Z 468.912,A -85,B 0,C 180,E1 -19446.659,E2 -19446.659} C_VEL
LIN {X 0,Y 242.336,Z 468.894,A -85,B 0,C 180,E1 -19450.021,E2 -19450.021} C_VEL
LIN {X 0,Y 242.158,Z 468.941,A -85,B 0,C 180,E1 -19455.141,E2 -19455.141} C_VEL
LIN {X 0,Y 242.063,Z 468.936,A -85,B 0,C 180,E1 -19458.625,E2 -19458.625} C_VEL
LIN {X 0,Y 242.004,Z 468.96,A -85,B 0,C 180,E1 -19462.181,E2 -19462.181} C_VEL
LIN {X 0,Y 242.057,Z 468.955,A -85,B 0,C 180,E1 -19465.839,E2 -19465.839} C_VEL
LIN {X 0,Y 242.022,Z 468.965,A -85,B 0,C 180,E1 -19469.581,E2 -19469.581} C_VEL
LIN {X 0,Y 241.964,Z 468.968,A -85,B 0,C 180,E1 -19471.903,E2 -19471.903} C_VEL
LIN {X 0,Y 241.319,Z 469.053,A -85,B 0,C 180,E1 -19473.294,E2 -19473.294} C_VEL
LIN {X 0,Y 238.508,Z 469.407,A -85,B 0,C 180,E1 -19475.562,E2 -19475.562} C_VEL
LIN {X 0,Y 236.096,Z 469.704,A -85,B 0,C 180,E1 -19477.411,E2 -19477.411} C_VEL
LIN {X 0,Y 235.037,Z 469.83,A -85,B 0,C 180,E1 -19478.844,E2 -19478.844} C_VEL
LIN {X 0,Y 234.938,Z 469.839,A -85,B 0,C 180,E1 -19479.33,E2 -19479.33} C_VEL
LIN {X 0,Y 235.068,Z 469.96,A -85,B 0,C 180,E1 -19481.951,E2 -19481.951} C_VEL
LIN {X 0,Y 237.033,Z 478.369,A -85,B 0,C 180,E1 -19485.949,E2 -19485.949} C_VEL
LIN {X 0,Y 239.215,Z 487.264,A -85,B 0,C 180,E1 -19489.806,E2 -19489.806} C_VEL
LIN {X 0,Y 240.449,Z 492.54,A -85,B 0,C 180,E1 -19491.828,E2 -19491.828} C_VEL
LIN {X 0,Y 245.332,Z 502.468,A -85,B 0,C 180,E1 -19493.097,E2 -19493.097} C_VEL
LIN {X 0,Y 248.833,Z 515.254,A -85,B 0,C 180,E1 -19494.388,E2 -19494.388} C_VEL
LIN {X 0,Y 250.958,Z 527.721,A -85,B 0,C 180,E1 -19495.706,E2 -19495.706} C_VEL
LIN {X 0,Y 252.181,Z 541.016,A -85,B 0,C 180,E1 -19497.276,E2 -19497.276} C_VEL
LIN {X 0,Y 252.571,Z 553.789,A -85,B 0,C 180,E1 -19499.02,E2 -19499.02} C_VEL
LIN {X 0,Y 251.873,Z 558.361,A -85,B 0,C 180,E1 -19499.622,E2 -19499.622} C_VEL
LIN {X 0,Y 249.112,Z 570.139,A -85,B 0,C 180,E1 -19501.343,E2 -19501.343} C_VEL
LIN {X 0,Y 246.217,Z 580.893,A -85,B 0,C 180,E1 -19503.287,E2 -19503.287} C_VEL
LIN {X 0,Y 243.527,Z 589.895,A -85,B 0,C 180,E1 -19505.265,E2 -19505.265} C_VEL
LIN {X 0,Y 240.783,Z 598.918,A -85,B 0,C 180,E1 -19507.703,E2 -19507.703} C_VEL
LIN {X 0,Y 238.087,Z 607.532,A -85,B 0,C 180,E1 -19510.607,E2 -19510.607} C_VEL
LIN {X 0,Y 236.14,Z 614.468,A -85,B 0,C 180,E1 -19513.579,E2 -19513.579} C_VEL
LIN {X 0,Y 234.698,Z 619.258,A -85,B 0,C 180,E1 -19516.142,E2 -19516.142} C_VEL
LIN {X 0,Y 233.519,Z 624.2,A -85,B 0,C 180,E1 -19519.599,E2 -19519.599} C_VEL
LIN {X 0,Y 232.886,Z 627.633,A -85,B 0,C 180,E1 -19523.069,E2 -19523.069} C_VEL
LIN {X 0,Y 232.683,Z 629.661,A -85,B 0,C 180,E1 -19526.539,E2 -19526.539} C_VEL
LIN {X 0,Y 232.714,Z 630.165,A -85,B 0,C 180,E1 -19528.272,E2 -19528.272} C_VEL
LIN {X 0,Y 232.739,Z 630.329,A -85,B 0,C 180,E1 -19530.002,E2 -19530.002} C_VEL
LIN {X 0,Y 232.715,Z 630.155,A -85,B 0,C 180,E1 -19531.733,E2 -19531.733} C_VEL
LIN {X 0,Y 232.745,Z 628.789,A -85,B 0,C 180,E1 -19535.2,E2 -19535.2} C_VEL
LIN {X 0,Y 233.123,Z 626.051,A -85,B 0,C 180,E1 -19538.672,E2 -19538.672} C_VEL
LIN {X 0,Y 234.031,Z 621.867,A -85,B 0,C 180,E1 -19542.137,E2 -19542.137} C_VEL
LIN {X 0,Y 235.173,Z 617.713,A -85,B 0,C 180,E1 -19544.717,E2 -19544.717} C_VEL
LIN {X 0,Y 235.672,Z 616.105,A -85,B 0,C 180,E1 -19545.571,E2 -19545.571} C_VEL
LIN {X 0,Y 238.602,Z 611.634,A -85,B 0,C 180,E1 -19549.514,E2 -19549.514} C_VEL
LIN {X 0,Y 242.694,Z 606.212,A -85,B 0,C 180,E1 -19553.015,E2 -19553.015} C_VEL
LIN {X 0,Y 247.3,Z 599.858,A -85,B 0,C 180,E1 -19556.137,E2 -19556.137} C_VEL
LIN {X 0,Y 252.898,Z 592.059,A -85,B 0,C 180,E1 -19559.101,E2 -19559.101} C_VEL
LIN {X 0,Y 259.474,Z 582.622,A -85,B 0,C 180,E1 -19561.884,E2 -19561.884} C_VEL
LIN {X 0,Y 265.943,Z 572.857,A -85,B 0,C 180,E1 -19564.166,E2 -19564.166} C_VEL
LIN {X 0,Y 269.647,Z 566.879,A -85,B 0,C 180,E1 -19565.375,E2 -19565.375} C_VEL
LIN {X 0,Y 271.712,Z 561.228,A -85,B 0,C 180,E1 -19566.97,E2 -19566.97} C_VEL
LIN {X 0,Y 273.644,Z 554.706,A -85,B 0,C 180,E1 -19569.041,E2 -19569.041} C_VEL
LIN {X 0,Y 273.978,Z 552.671,A -85,B 0,C 180,E1 -19569.89,E2 -19569.89} C_VEL
LIN {X 0,Y 274.005,Z 551.209,A -85,B 0,C 180,E1 -19570.713,E2 -19570.713} C_VEL
LIN {X 0,Y 273.85,Z 549.562,A -85,B 0,C 180,E1 -19571.906,E2 -19571.906} C_VEL
LIN {X 0,Y 273.495,Z 547.668,A -85,B 0,C 180,E1 -19573.985,E2 -19573.985} C_VEL
LIN {X 0,Y 273.207,Z 546.715,A -85,B 0,C 180,E1 -19576.079,E2 -19576.079} C_VEL
LIN {X 0,Y 273.172,Z 546.567,A -85,B 0,C 180,E1 -19578.255,E2 -19578.255} C_VEL
LIN {X 0,Y 273.096,Z 547.732,A -85,B 0,C 180,E1 -19580.539,E2 -19580.539} C_VEL
LIN {X 0,Y 272.916,Z 549.041,A -85,B 0,C 180,E1 -19581.827,E2 -19581.827} C_VEL
LIN {X 0,Y 272.172,Z 553.134,A -85,B 0,C 180,E1 -19584.432,E2 -19584.432} C_VEL
LIN {X 0,Y 271.304,Z 557.146,A -85,B 0,C 180,E1 -19586.401,E2 -19586.401} C_VEL
LIN {X 0,Y 270.225,Z 560.967,A -85,B 0,C 180,E1 -19588.018,E2 -19588.018} C_VEL
LIN {X 0,Y 268.293,Z 564.233,A -85,B 0,C 180,E1 -19588.845,E2 -19588.845} C_VEL
LIN {X 0,Y 261.941,Z 573.071,A -85,B 0,C 180,E1 -19591.122,E2 -19591.122} C_VEL
LIN {X 0,Y 257.01,Z 579.524,A -85,B 0,C 180,E1 -19593.18,E2 -19593.18} C_VEL
LIN {X 0,Y 251.035,Z 586.637,A -85,B 0,C 180,E1 -19596.05,E2 -19596.05} C_VEL
LIN {X 0,Y 247.224,Z 590.877,A -85,B 0,C 180,E1 -19598.312,E2 -19598.312} C_VEL
LIN {X 0,Y 242.863,Z 595.311,A -85,B 0,C 180,E1 -19601.439,E2 -19601.439} C_VEL
LIN {X 0,Y 239.229,Z 598.321,A -85,B 0,C 180,E1 -19604.669,E2 -19604.669} C_VEL
LIN {X 0,Y 236.719,Z 599.972,A -85,B 0,C 180,E1 -19608.005,E2 -19608.005} C_VEL
LIN {X 0,Y 234.705,Z 600.295,A -85,B 0,C 180,E1 -19611.389,E2 -19611.389} C_VEL
LIN {X 0,Y 233.601,Z 599.204,A -85,B 0,C 180,E1 -19614.822,E2 -19614.822} C_VEL
LIN {X 0,Y 233.082,Z 596.642,A -85,B 0,C 180,E1 -19618.272,E2 -19618.272} C_VEL
LIN {X 0,Y 232.982,Z 592.553,A -85,B 0,C 180,E1 -19621.729,E2 -19621.729} C_VEL
LIN {X 0,Y 233.011,Z 588.361,A -85,B 0,C 180,E1 -19624.325,E2 -19624.325} C_VEL
LIN {X 0,Y 233.299,Z 583.128,A -85,B 0,C 180,E1 -19626.921,E2 -19626.921} C_VEL
LIN {X 0,Y 233.787,Z 576.686,A -85,B 0,C 180,E1 -19629.517,E2 -19629.517} C_VEL
LIN {X 0,Y 234.641,Z 568.878,A -85,B 0,C 180,E1 -19632.103,E2 -19632.103} C_VEL
LIN {X 0,Y 235.719,Z 559.382,A -85,B 0,C 180,E1 -19634.681,E2 -19634.681} C_VEL
LIN {X 0,Y 237.222,Z 547.906,A -85,B 0,C 180,E1 -19637.233,E2 -19637.233} C_VEL
LIN {X 0,Y 238.621,Z 536.979,A -85,B 0,C 180,E1 -19639.216,E2 -19639.216} C_VEL
LIN {X 0,Y 239.96,Z 526.501,A -85,B 0,C 180,E1 -19640.801,E2 -19640.801} C_VEL
LIN {X 0,Y 238.87,Z 517.453,A -85,B 0,C 180,E1 -19642.032,E2 -19642.032} C_VEL
LIN {X 0,Y 236.703,Z 503.106,A -85,B 0,C 180,E1 -19643.673,E2 -19643.673} C_VEL
LIN {X 0,Y 234.479,Z 488.97,A -85,B 0,C 180,E1 -19644.958,E2 -19644.958} C_VEL
LIN {X 0,Y 234.059,Z 485.609,A -85,B 0,C 180,E1 -19645.228,E2 -19645.228} C_VEL
LIN {X 0,Y 234.63,Z 480.669,A -85,B 0,C 180,E1 -19649.694,E2 -19649.694} C_VEL
LIN {X 0,Y 235.123,Z 476.9,A -85,B 0,C 180,E1 -19653.179,E2 -19653.179} C_VEL
LIN {X 0,Y 235.341,Z 473.434,A -85,B 0,C 180,E1 -19656.514,E2 -19656.514} C_VEL
LIN {X 0,Y 236.644,Z 476.736,A -85,B 0,C 180,E1 -19659.449,E2 -19659.449} C_VEL
LIN {X 0,Y 237.662,Z 482.33,A -85,B 0,C 180,E1 -19663.862,E2 -19663.862} C_VEL
LIN {X 0,Y 238.489,Z 487.167,A -85,B 0,C 180,E1 -19667.453,E2 -19667.453} C_VEL
LIN {X 0,Y 238.808,Z 490.736,A -85,B 0,C 180,E1 -19669.922,E2 -19669.922} C_VEL
LIN {X 0,Y 238.646,Z 493.335,A -85,B 0,C 180,E1 -19671.481,E2 -19671.481} C_VEL
LIN {X 0,Y 240.039,Z 496.854,A -85,B 0,C 180,E1 -19671.88,E2 -19671.88} C_VEL
LIN {X 0,Y 245.182,Z 510.888,A -85,B 0,C 180,E1 -19673.557,E2 -19673.557} C_VEL
LIN {X 0,Y 248.562,Z 523.063,A -85,B 0,C 180,E1 -19675.082,E2 -19675.082} C_VEL
LIN {X 0,Y 250.913,Z 535.153,A -85,B 0,C 180,E1 -19676.693,E2 -19676.693} C_VEL
LIN {X 0,Y 252.384,Z 547.729,A -85,B 0,C 180,E1 -19678.524,E2 -19678.524} C_VEL
LIN {X 0,Y 252.622,Z 554.559,A -85,B 0,C 180,E1 -19679.591,E2 -19679.591} C_VEL
LIN {X 0,Y 249.687,Z 566.927,A -85,B 0,C 180,E1 -19681.41,E2 -19681.41} C_VEL
LIN {X 0,Y 246.693,Z 577.555,A -85,B 0,C 180,E1 -19683.338,E2 -19683.338} C_VEL
LIN {X 0,Y 243.624,Z 588.069,A -85,B 0,C 180,E1 -19685.725,E2 -19685.725} C_VEL
LIN {X 0,Y 240.894,Z 596.748,A -85,B 0,C 180,E1 -19688.16,E2 -19688.16} C_VEL
LIN {X 0,Y 238.287,Z 605.06,A -85,B 0,C 180,E1 -19691.067,E2 -19691.067} C_VEL
LIN {X 0,Y 236.617,Z 610.848,A -85,B 0,C 180,E1 -19693.608,E2 -19693.608} C_VEL
LIN {X 0,Y 234.714,Z 617.021,A -85,B 0,C 180,E1 -19697.02,E2 -19697.02} C_VEL
LIN {X 0,Y 233.763,Z 620.526,A -85,B 0,C 180,E1 -19699.606,E2 -19699.606} C_VEL
LIN {X 0,Y 232.998,Z 623.946,A -85,B 0,C 180,E1 -19703.068,E2 -19703.068} C_VEL
LIN {X 0,Y 232.702,Z 625.98,A -85,B 0,C 180,E1 -19706.535,E2 -19706.535} C_VEL
LIN {X 0,Y 232.72,Z 626.676,A -85,B 0,C 180,E1 -19709.998,E2 -19709.998} C_VEL
LIN {X 0,Y 232.7,Z 626.04,A -85,B 0,C 180,E1 -19713.461,E2 -19713.461} C_VEL
LIN {X 0,Y 232.996,Z 624.058,A -85,B 0,C 180,E1 -19716.928,E2 -19716.928} C_VEL
LIN {X 0,Y 233.752,Z 620.687,A -85,B 0,C 180,E1 -19720.391,E2 -19720.391} C_VEL
LIN {X 0,Y 234.984,Z 615.826,A -85,B 0,C 180,E1 -19723.841,E2 -19723.841} C_VEL
LIN {X 0,Y 237.179,Z 609.329,A -85,B 0,C 180,E1 -19727.234,E2 -19727.234} C_VEL
LIN {X 0,Y 239.082,Z 602.703,A -85,B 0,C 180,E1 -19729.953,E2 -19729.953} C_VEL
LIN {X 0,Y 241.696,Z 594.475,A -85,B 0,C 180,E1 -19732.659,E2 -19732.659} C_VEL
LIN {X 0,Y 244.519,Z 585.335,A -85,B 0,C 180,E1 -19735.081,E2 -19735.081} C_VEL
LIN {X 0,Y 247.513,Z 575.212,A -85,B 0,C 180,E1 -19737.247,E2 -19737.247} C_VEL
LIN {X 0,Y 250.647,Z 563.44,A -85,B 0,C 180,E1 -19739.266,E2 -19739.266} C_VEL
LIN {X 0,Y 252.761,Z 553.891,A -85,B 0,C 180,E1 -19740.632,E2 -19740.632} C_VEL
LIN {X 0,Y 252.006,Z 543.148,A -85,B 0,C 180,E1 -19742.29,E2 -19742.29} C_VEL
LIN {X 0,Y 250.203,Z 530.69,A -85,B 0,C 180,E1 -19744.043,E2 -19744.043} C_VEL
LIN {X 0,Y 247.123,Z 517.333,A -85,B 0,C 180,E1 -19745.78,E2 -19745.78} C_VEL
LIN {X 0,Y 242.77,Z 503.812,A -85,B 0,C 180,E1 -19747.437,E2 -19747.437} C_VEL
LIN {X 0,Y 238.703,Z 493.432,A -85,B 0,C 180,E1 -19748.65,E2 -19748.65} C_VEL
LIN {X 0,Y 238.69,Z 492.726,A -85,B 0,C 180,E1 -19748.943,E2 -19748.943} C_VEL
LIN {X 0,Y 238.791,Z 488.98,A -85,B 0,C 180,E1 -19751.434,E2 -19751.434} C_VEL
LIN {X 0,Y 238.007,Z 483.902,A -85,B 0,C 180,E1 -19755.124,E2 -19755.124} C_VEL
LIN {X 0,Y 236.968,Z 478.541,A -85,B 0,C 180,E1 -19759.271,E2 -19759.271} C_VEL
LIN {X 0,Y 235.852,Z 473.59,A -85,B 0,C 180,E1 -19763.418,E2 -19763.418} C_VEL
LIN {X 0,Y 234.954,Z 469.844,A -85,B 0,C 180,E1 -19766.877,E2 -19766.877} C_VEL
LIN {X 0,Y 234.946,Z 469.845,A -85,B 0,C 180,E1 -19771.405,E2 -19771.405} C_VEL
LIN {X 0,Y 234.983,Z 469.84,A -85,B 0,C 180,E1 -19775.246,E2 -19775.246} C_VEL
LIN {X 0,Y 235.034,Z 469.817,A -85,B 0,C 180,E1 -19778.972,E2 -19778.972} C_VEL
LIN {X 0,Y 235.107,Z 469.823,A -85,B 0,C 180,E1 -19783.042,E2 -19783.042} C_VEL
LIN {X 0,Y 235.138,Z 469.814,A -85,B 0,C 180,E1 -19787.923,E2 -19787.923} C_VEL
LIN {X 0,Y 235.381,Z 469.783,A -85,B 0,C 180,E1 -19791.414,E2 -19791.414} C_VEL
LIN {X 0,Y 235.397,Z 469.789,A -85,B 0,C 180,E1 -19793.141,E2 -19793.141} C_VEL
LIN {X 0,Y 235.595,Z 469.756,A -85,B 0,C 180,E1 -19798.29,E2 -19798.29} C_VEL
LIN {X 0,Y 235.587,Z 469.749,A -85,B 0,C 180,E1 -19801.709,E2 -19801.709} C_VEL
LIN {X 0,Y 235.396,Z 469.789,A -85,B 0,C 180,E1 -19806.859,E2 -19806.859} C_VEL
LIN {X 0,Y 235.244,Z 469.776,A -85,B 0,C 180,E1 -19810.326,E2 -19810.326} C_VEL
LIN {X 0,Y 235.104,Z 469.811,A -85,B 0,C 180,E1 -19815.607,E2 -19815.607} C_VEL
LIN {X 0,Y 234.999,Z 469.822,A -85,B 0,C 180,E1 -19819.206,E2 -19819.206} C_VEL
LIN {X 0,Y 234.952,Z 469.84,A -85,B 0,C 180,E1 -19822.884,E2 -19822.884} C_VEL
LIN {X 0,Y 234.961,Z 469.844,A -85,B 0,C 180,E1 -19826.658,E2 -19826.658} C_VEL
LIN {X 0,Y 234.924,Z 469.845,A -85,B 0,C 180,E1 -19830.569,E2 -19830.569} C_VEL
LIN {X 0,Y 234.952,Z 469.843,A -85,B 0,C 180,E1 -19834.634,E2 -19834.634} C_VEL
LIN {X 0,Y 234.938,Z 469.839,A -85,B 0,C 180,E1 -19839.33,E2 -19839.33} C_VEL
LIN {X 0,Y 234.692,Z 470.228,A -85,B 0,C 180,E1 -19840.276,E2 -19840.276} C_VEL
LIN {X 0,Y 233.788,Z 471.958,A -85,B 0,C 180,E1 -19841.639,E2 -19841.639} C_VEL
LIN {X 0,Y 232.627,Z 474.582,A -85,B 0,C 180,E1 -19842.922,E2 -19842.922} C_VEL
LIN {X 0,Y 231.298,Z 478.862,A -85,B 0,C 180,E1 -19844.614,E2 -19844.614} C_VEL
LIN {X 0,Y 231.038,Z 482.079,A -85,B 0,C 180,E1 -19845.901,E2 -19845.901} C_VEL
LIN {X 0,Y 231.18,Z 483.07,A -85,B 0,C 180,E1 -19846.34,E2 -19846.34} C_VEL
LIN {X 0,Y 233.289,Z 492.271,A -85,B 0,C 180,E1 -19850.401,E2 -19850.401} C_VEL
LIN {X 0,Y 239.939,Z 505.593,A -85,B 0,C 180,E1 -19852.265,E2 -19852.265} C_VEL
LIN {X 0,Y 243.122,Z 517.792,A -85,B 0,C 180,E1 -19853.6,E2 -19853.6} C_VEL
LIN {X 0,Y 244.92,Z 529.042,A -85,B 0,C 180,E1 -19854.868,E2 -19854.868} C_VEL
LIN {X 0,Y 245.998,Z 541.87,A -85,B 0,C 180,E1 -19856.455,E2 -19856.455} C_VEL
LIN {X 0,Y 246.233,Z 553.754,A -85,B 0,C 180,E1 -19858.13,E2 -19858.13} C_VEL
LIN {X 0,Y 245.771,Z 558.325,A -85,B 0,C 180,E1 -19858.785,E2 -19858.785} C_VEL
LIN {X 0,Y 242.892,Z 570.098,A -85,B 0,C 180,E1 -19860.538,E2 -19860.538} C_VEL
LIN {X 0,Y 239.886,Z 580.848,A -85,B 0,C 180,E1 -19862.523,E2 -19862.523} C_VEL
LIN {X 0,Y 237.072,Z 589.847,A -85,B 0,C 180,E1 -19864.544,E2 -19864.544} C_VEL
LIN {X 0,Y 234.21,Z 598.868,A -85,B 0,C 180,E1 -19867.042,E2 -19867.042} C_VEL
LIN {X 0,Y 231.365,Z 607.48,A -85,B 0,C 180,E1 -19870.02,E2 -19870.02} C_VEL
LIN {X 0,Y 229.271,Z 614.415,A -85,B 0,C 180,E1 -19873.072,E2 -19873.072} C_VEL
LIN {X 0,Y 227.787,Z 619.205,A -85,B 0,C 180,E1 -19875.713,E2 -19875.713} C_VEL
LIN {X 0,Y 226.511,Z 624.146,A -85,B 0,C 180,E1 -19879.273,E2 -19879.273} C_VEL
LIN {X 0,Y 225.814,Z 627.578,A -85,B 0,C 180,E1 -19882.851,E2 -19882.851} C_VEL
LIN {X 0,Y 225.599,Z 629.606,A -85,B 0,C 180,E1 -19886.43,E2 -19886.43} C_VEL
LIN {X 0,Y 225.655,Z 630.274,A -85,B 0,C 180,E1 -19890.002,E2 -19890.002} C_VEL
LIN {X 0,Y 225.601,Z 629.585,A -85,B 0,C 180,E1 -19893.574,E2 -19893.574} C_VEL
LIN {X 0,Y 225.816,Z 627.539,A -85,B 0,C 180,E1 -19897.154,E2 -19897.154} C_VEL
LIN {X 0,Y 226.511,Z 624.091,A -85,B 0,C 180,E1 -19900.731,E2 -19900.731} C_VEL
LIN {X 0,Y 227.778,Z 619.136,A -85,B 0,C 180,E1 -19904.293,E2 -19904.293} C_VEL
LIN {X 0,Y 228.924,Z 615.822,A -85,B 0,C 180,E1 -19906.271,E2 -19906.271} C_VEL
LIN {X 0,Y 231.769,Z 612.269,A -85,B 0,C 180,E1 -19909.945,E2 -19909.945} C_VEL
LIN {X 0,Y 236.229,Z 606.992,A -85,B 0,C 180,E1 -19913.683,E2 -19913.683} C_VEL
LIN {X 0,Y 241.043,Z 601.008,A -85,B 0,C 180,E1 -19916.869,E2 -19916.869} C_VEL
LIN {X 0,Y 246.89,Z 593.657,A -85,B 0,C 180,E1 -19919.88,E2 -19919.88} C_VEL
LIN {X 0,Y 253.702,Z 584.812,A -85,B 0,C 180,E1 -19922.698,E2 -19922.698} C_VEL
LIN {X 0,Y 260.407,Z 575.638,A -85,B 0,C 180,E1 -19924.997,E2 -19924.997} C_VEL
LIN {X 0,Y 264.339,Z 569.932,A -85,B 0,C 180,E1 -19926.196,E2 -19926.196} C_VEL
LIN {X 0,Y 266.268,Z 565.824,A -85,B 0,C 180,E1 -19927.38,E2 -19927.38} C_VEL
LIN {X 0,Y 268.569,Z 559.698,A -85,B 0,C 180,E1 -19929.414,E2 -19929.414} C_VEL
LIN {X 0,Y 268.938,Z 558.538,A -85,B 0,C 180,E1 -19929.858,E2 -19929.858} C_VEL
LIN {X 0,Y 269.267,Z 556.672,A -85,B 0,C 180,E1 -19930.807,E2 -19930.807} C_VEL
LIN {X 0,Y 269.123,Z 554.29,A -85,B 0,C 180,E1 -19932.766,E2 -19932.766} C_VEL
LIN {X 0,Y 268.835,Z 552.672,A -85,B 0,C 180,E1 -19935.102,E2 -19935.102} C_VEL
LIN {X 0,Y 268.689,Z 552.133,A -85,B 0,C 180,E1 -19937.151,E2 -19937.151} C_VEL
LIN {X 0,Y 268.608,Z 552.56,A -85,B 0,C 180,E1 -19939.358,E2 -19939.358} C_VEL
LIN {X 0,Y 268.348,Z 553.768,A -85,B 0,C 180,E1 -19941.056,E2 -19941.056} C_VEL
LIN {X 0,Y 267.462,Z 557.007,A -85,B 0,C 180,E1 -19943.492,E2 -19943.492} C_VEL
LIN {X 0,Y 266.239,Z 561.162,A -85,B 0,C 180,E1 -19945.779,E2 -19945.779} C_VEL
LIN {X 0,Y 265.246,Z 564.086,A -85,B 0,C 180,E1 -19947.1,E2 -19947.1} C_VEL
LIN {X 0,Y 264.62,Z 565.166,A -85,B 0,C 180,E1 -19947.465,E2 -19947.465} C_VEL
LIN {X 0,Y 257.05,Z 574.979,A -85,B 0,C 180,E1 -19950.068,E2 -19950.068} C_VEL
LIN {X 0,Y 251.022,Z 582.019,A -85,B 0,C 180,E1 -19952.486,E2 -19952.486} C_VEL
LIN {X 0,Y 244.8,Z 588.639,A -85,B 0,C 180,E1 -19955.4,E2 -19955.4} C_VEL
LIN {X 0,Y 239.612,Z 593.731,A -85,B 0,C 180,E1 -19958.492,E2 -19958.492} C_VEL
LIN {X 0,Y 236.265,Z 596.599,A -85,B 0,C 180,E1 -19960.901,E2 -19960.901} C_VEL
LIN {X 0,Y 232.469,Z 599.32,A -85,B 0,C 180,E1 -19964.212,E2 -19964.212} C_VEL
LIN {X 0,Y 229.819,Z 600.665,A -85,B 0,C 180,E1 -19967.64,E2 -19967.64} C_VEL
LIN {X 0,Y 227.719,Z 600.675,A -85,B 0,C 180,E1 -19971.123,E2 -19971.123} C_VEL
LIN {X 0,Y 226.525,Z 599.29,A -85,B 0,C 180,E1 -19974.66,E2 -19974.66} C_VEL
LIN {X 0,Y 226.015,Z 596.487,A -85,B 0,C 180,E1 -19978.218,E2 -19978.218} C_VEL
LIN {X 0,Y 225.882,Z 593.379,A -85,B 0,C 180,E1 -19980.892,E2 -19980.892} C_VEL
LIN {X 0,Y 225.929,Z 589.325,A -85,B 0,C 180,E1 -19983.567,E2 -19983.567} C_VEL
LIN {X 0,Y 226.097,Z 584.218,A -85,B 0,C 180,E1 -19986.245,E2 -19986.245} C_VEL
LIN {X 0,Y 226.671,Z 576.808,A -85,B 0,C 180,E1 -19989.368,E2 -19989.368} C_VEL
LIN {X 0,Y 227.482,Z 569.023,A -85,B 0,C 180,E1 -19992.037,E2 -19992.037} C_VEL
LIN {X 0,Y 228.587,Z 559.504,A -85,B 0,C 180,E1 -19994.694,E2 -19994.694} C_VEL
LIN {X 0,Y 229.955,Z 549.014,A -85,B 0,C 180,E1 -19997.108,E2 -19997.108} C_VEL
LIN {X 0,Y 231.318,Z 538.8,A -85,B 0,C 180,E1 -19999.063,E2 -19999.063} C_VEL
LIN {X 0,Y 232.907,Z 526.25,A -85,B 0,C 180,E1 -20001.035,E2 -20001.035} C_VEL
LIN {X 0,Y 231.07,Z 513.15,A -85,B 0,C 180,E1 -20002.817,E2 -20002.817} C_VEL
LIN {X 0,Y 228.913,Z 499.315,A -85,B 0,C 180,E1 -20004.35,E2 -20004.35} C_VEL
LIN {X 0,Y 227.015,Z 485.795,A -85,B 0,C 180,E1 -20005.562,E2 -20005.562} C_VEL
LIN {X 0,Y 227.634,Z 480.814,A -85,B 0,C 180,E1 -20010.174,E2 -20010.174} C_VEL
LIN {X 0,Y 228.087,Z 477.12,A -85,B 0,C 180,E1 -20013.698,E2 -20013.698} C_VEL
LIN {X 0,Y 228.211,Z 475.114,A -85,B 0,C 180,E1 -20015.744,E2 -20015.744} C_VEL
LIN {X 0,Y 229.735,Z 478.368,A -85,B 0,C 180,E1 -20018.839,E2 -20018.839} C_VEL
LIN {X 0,Y 230.721,Z 483.487,A -85,B 0,C 180,E1 -20023.022,E2 -20023.022} C_VEL
LIN {X 0,Y 231.547,Z 488.37,A -85,B 0,C 180,E1 -20026.757,E2 -20026.757} C_VEL
LIN {X 0,Y 232.02,Z 492.159,A -85,B 0,C 180,E1 -20029.494,E2 -20029.494} C_VEL
LIN {X 0,Y 231.991,Z 493.351,A -85,B 0,C 180,E1 -20030.163,E2 -20030.163} C_VEL
LIN {X 0,Y 237.545,Z 507.591,A -85,B 0,C 180,E1 -20031.973,E2 -20031.973} C_VEL
LIN {X 0,Y 241.663,Z 521.174,A -85,B 0,C 180,E1 -20033.762,E2 -20033.762} C_VEL
LIN {X 0,Y 244.227,Z 533.464,A -85,B 0,C 180,E1 -20035.459,E2 -20035.459} C_VEL
LIN {X 0,Y 245.828,Z 546.055,A -85,B 0,C 180,E1 -20037.34,E2 -20037.34} C_VEL
LIN {X 0,Y 246.291,Z 555.509,A -85,B 0,C 180,E1 -20038.877,E2 -20038.877} C_VEL
LIN {X 0,Y 243.139,Z 568.128,A -85,B 0,C 180,E1 -20040.803,E2 -20040.803} C_VEL
LIN {X 0,Y 239.769,Z 579.525,A -85,B 0,C 180,E1 -20042.976,E2 -20042.976} C_VEL
LIN {X 0,Y 236.68,Z 589.722,A -85,B 0,C 180,E1 -20045.433,E2 -20045.433} C_VEL
LIN {X 0,Y 233.848,Z 598.133,A -85,B 0,C 180,E1 -20047.932,E2 -20047.932} C_VEL
LIN {X 0,Y 231.221,Z 606.158,A -85,B 0,C 180,E1 -20050.926,E2 -20050.926} C_VEL
LIN {X 0,Y 229.798,Z 610.903,A -85,B 0,C 180,E1 -20053.107,E2 -20053.107} C_VEL
LIN {X 0,Y 227.755,Z 617.077,A -85,B 0,C 180,E1 -20056.616,E2 -20056.616} C_VEL
LIN {X 0,Y 226.765,Z 620.582,A -85,B 0,C 180,E1 -20059.281,E2 -20059.281} C_VEL
LIN {X 0,Y 225.936,Z 624.003,A -85,B 0,C 180,E1 -20062.85,E2 -20062.85} C_VEL
LIN {X 0,Y 225.617,Z 626.036,A -85,B 0,C 180,E1 -20066.426,E2 -20066.426} C_VEL
LIN {X 0,Y 225.636,Z 626.732,A -85,B 0,C 180,E1 -20069.998,E2 -20069.998} C_VEL
LIN {X 0,Y 225.614,Z 626.096,A -85,B 0,C 180,E1 -20073.57,E2 -20073.57} C_VEL
LIN {X 0,Y 225.934,Z 624.113,A -85,B 0,C 180,E1 -20077.145,E2 -20077.145} C_VEL
LIN {X 0,Y 226.752,Z 620.742,A -85,B 0,C 180,E1 -20080.715,E2 -20080.715} C_VEL
LIN {X 0,Y 228.061,Z 615.88,A -85,B 0,C 180,E1 -20084.27,E2 -20084.27} C_VEL
LIN {X 0,Y 230.347,Z 609.381,A -85,B 0,C 180,E1 -20087.762,E2 -20087.762} C_VEL
LIN {X 0,Y 232.622,Z 602.026,A -85,B 0,C 180,E1 -20090.834,E2 -20090.834} C_VEL
LIN {X 0,Y 235.628,Z 593.096,A -85,B 0,C 180,E1 -20093.742,E2 -20093.742} C_VEL
LIN {X 0,Y 238.614,Z 583.639,A -85,B 0,C 180,E1 -20096.216,E2 -20096.216} C_VEL
LIN {X 0,Y 241.811,Z 573.154,A -85,B 0,C 180,E1 -20098.417,E2 -20098.417} C_VEL
LIN {X 0,Y 244.815,Z 562.115,A -85,B 0,C 180,E1 -20100.29,E2 -20100.29} C_VEL
LIN {X 0,Y 246.407,Z 554.79,A -85,B 0,C 180,E1 -20101.365,E2 -20101.365} C_VEL
LIN {X 0,Y 245.554,Z 542.842,A -85,B 0,C 180,E1 -20103.294,E2 -20103.294} C_VEL
LIN {X 0,Y 243.731,Z 530.233,A -85,B 0,C 180,E1 -20105.132,E2 -20105.132} C_VEL
LIN {X 0,Y 240.477,Z 516.704,A -85,B 0,C 180,E1 -20106.981,E2 -20106.981} C_VEL
LIN {X 0,Y 236.122,Z 503.636,A -85,B 0,C 180,E1 -20108.689,E2 -20108.689} C_VEL
LIN {X 0,Y 232.022,Z 493.121,A -85,B 0,C 180,E1 -20110.027,E2 -20110.027} C_VEL
LIN {X 0,Y 231.941,Z 490.56,A -85,B 0,C 180,E1 -20111.803,E2 -20111.803} C_VEL
LIN {X 0,Y 231.131,Z 485.411,A -85,B 0,C 180,E1 -20115.624,E2 -20115.624} C_VEL
LIN {X 0,Y 230.133,Z 480.306,A -85,B 0,C 180,E1 -20119.767,E2 -20119.767} C_VEL
LIN {X 0,Y 229.375,Z 476.739,A -85,B 0,C 180,E1 -20122.806,E2 -20122.806} C_VEL
LIN {X 0,Y 228.107,Z 471.703,A -85,B 0,C 180,E1 -20127.372,E2 -20127.372} C_VEL
LIN {X 0,Y 227.865,Z 470.718,A -85,B 0,C 180,E1 -20128.377,E2 -20128.377} C_VEL
LIN {X 0,Y 227.88,Z 470.713,A -85,B 0,C 180,E1 -20132.444,E2 -20132.444} C_VEL
LIN {X 0,Y 227.922,Z 470.712,A -85,B 0,C 180,E1 -20136.368,E2 -20136.368} C_VEL
LIN {X 0,Y 227.956,Z 470.713,A -85,B 0,C 180,E1 -20140.176,E2 -20140.176} C_VEL
LIN {X 0,Y 228.056,Z 470.703,A -85,B 0,C 180,E1 -20143.898,E2 -20143.898} C_VEL
LIN {X 0,Y 228.162,Z 470.688,A -85,B 0,C 180,E1 -20149.349,E2 -20149.349} C_VEL
LIN {X 0,Y 228.35,Z 470.667,A -85,B 0,C 180,E1 -20152.928,E2 -20152.928} C_VEL
LIN {X 0,Y 228.554,Z 470.633,A -85,B 0,C 180,E1 -20158.238,E2 -20158.238} C_VEL
LIN {X 0,Y 228.545,Z 470.624,A -85,B 0,C 180,E1 -20161.762,E2 -20161.762} C_VEL
LIN {X 0,Y 228.348,Z 470.667,A -85,B 0,C 180,E1 -20167.072,E2 -20167.072} C_VEL
LIN {X 0,Y 228.162,Z 470.657,A -85,B 0,C 180,E1 -20170.65,E2 -20170.65} C_VEL
LIN {X 0,Y 228.072,Z 470.701,A -85,B 0,C 180,E1 -20174.271,E2 -20174.271} C_VEL
LIN {X 0,Y 227.994,Z 470.682,A -85,B 0,C 180,E1 -20177.954,E2 -20177.954} C_VEL
LIN {X 0,Y 227.921,Z 470.714,A -85,B 0,C 180,E1 -20182.33,E2 -20182.33} C_VEL
LIN {X 0,Y 227.934,Z 470.719,A -85,B 0,C 180,E1 -20186.604,E2 -20186.604} C_VEL
LIN {X 0,Y 227.9,Z 470.721,A -85,B 0,C 180,E1 -20190.297,E2 -20190.297} C_VEL
LIN {X 0,Y 227.881,Z 470.721,A -85,B 0,C 180,E1 -20193.72,E2 -20193.72} C_VEL
LIN {X 0,Y 227.864,Z 470.727,A -85,B 0,C 180,E1 -20198.087,E2 -20198.087} C_VEL
LIN {X 0,Y 227.923,Z 470.874,A -85,B 0,C 180,E1 -20199.999,E2 -20199.999} C_VEL
LIN {X 0,Y 229.432,Z 475.588,A -85,B 0,C 180,E1 -20202.682,E2 -20202.682} C_VEL
LIN {X 0,Y 231.1,Z 482.704,A -85,B 0,C 180,E1 -20206.172,E2 -20206.172} C_VEL
LIN {X 0,Y 231.18,Z 483.07,A -85,B 0,C 180,E1 -20206.34,E2 -20206.34} C_VEL
LIN {X 0,Y 231.484,Z 486.469,A -85,B 0,C 180,E1 -20207.515,E2 -20207.515} C_VEL
LIN {X 0,Y 231.439,Z 490.758,A -85,B 0,C 180,E1 -20208.515,E2 -20208.515} C_VEL
LIN {X 0,Y 231.498,Z 497.21,A -85,B 0,C 180,E1 -20209.653,E2 -20209.653} C_VEL
LIN {X 0,Y 232.569,Z 503.886,A -85,B 0,C 180,E1 -20210.674,E2 -20210.674} C_VEL
LIN {X 0,Y 233.812,Z 507.056,A -85,B 0,C 180,E1 -20211.165,E2 -20211.165} C_VEL
LIN {X 0,Y 235.479,Z 511.713,A -85,B 0,C 180,E1 -20211.779,E2 -20211.779} C_VEL
LIN {X 0,Y 238.075,Z 523.796,A -85,B 0,C 180,E1 -20213.2,E2 -20213.2} C_VEL
LIN {X 0,Y 239.531,Z 537.097,A -85,B 0,C 180,E1 -20214.835,E2 -20214.835} C_VEL
LIN {X 0,Y 240.013,Z 550.514,A -85,B 0,C 180,E1 -20216.702,E2 -20216.702} C_VEL
LIN {X 0,Y 239.712,Z 558.288,A -85,B 0,C 180,E1 -20217.903,E2 -20217.903} C_VEL
LIN {X 0,Y 236.716,Z 570.056,A -85,B 0,C 180,E1 -20219.69,E2 -20219.69} C_VEL
LIN {X 0,Y 233.597,Z 580.803,A -85,B 0,C 180,E1 -20221.718,E2 -20221.718} C_VEL
LIN {X 0,Y 230.121,Z 591.418,A -85,B 0,C 180,E1 -20224.205,E2 -20224.205} C_VEL
LIN {X 0,Y 227.183,Z 600.167,A -85,B 0,C 180,E1 -20226.772,E2 -20226.772} C_VEL
LIN {X 0,Y 224.308,Z 608.541,A -85,B 0,C 180,E1 -20229.842,E2 -20229.842} C_VEL
LIN {X 0,Y 222.428,Z 614.362,A -85,B 0,C 180,E1 -20232.535,E2 -20232.535} C_VEL
LIN {X 0,Y 220.895,Z 619.151,A -85,B 0,C 180,E1 -20235.257,E2 -20235.257} C_VEL
LIN {X 0,Y 219.498,Z 624.091,A -85,B 0,C 180,E1 -20238.926,E2 -20238.926} C_VEL
LIN {X 0,Y 218.749,Z 627.523,A -85,B 0,C 180,E1 -20242.619,E2 -20242.619} C_VEL
LIN {X 0,Y 218.501,Z 629.55,A -85,B 0,C 180,E1 -20246.314,E2 -20246.314} C_VEL
LIN {X 0,Y 218.554,Z 630.218,A -85,B 0,C 180,E1 -20250.002,E2 -20250.002} C_VEL
